LIN {X 0,Y 474.637,Z 525.358,A -85,B 0,C 180,E1 -7446.642,E2 -7446.642} C_VEL
LIN {X 0,Y 474.66,Z 525.36,A -85,B 0,C 180,E1 -7450.09,E2 -7450.09} C_VEL
LIN {X 0,Y 474.663,Z 525.362,A -85,B 0,C 180,E1 -7451.685,E2 -7451.685} C_VEL
LIN {X 0,Y 474.409,Z 525.922,A -85,B 0,C 180,E1 -7452.155,E2 -7452.155} C_VEL
LIN {X 0,Y 473.767,Z 527.315,A -85,B 0,C 180,E1 -7452.599,E2 -7452.599} C_VEL
LIN {X 0,Y 471.839,Z 531.346,A -85,B 0,C 180,E1 -7453.425,E2 -7453.425} C_VEL
LIN {X 0,Y 469.145,Z 537.57,A -85,B 0,C 180,E1 -7454.637,E2 -7454.637} C_VEL
LIN {X 0,Y 468.823,Z 539.587,A -85,B 0,C 180,E1 -7455.057,E2 -7455.057} C_VEL
LIN {X 0,Y 468.432,Z 549.198,A -85,B 0,C 180,E1 -7457.076,E2 -7457.076} C_VEL
LIN {X 0,Y 471.299,Z 564.47,A -85,B 0,C 180,E1 -7457.416,E2 -7457.416} C_VEL
LIN {X 0,Y 470.623,Z 655.993,A -85,B 0,C 180,E1 -7458.833,E2 -7458.833} C_VEL
LIN {X 0,Y 470.332,Z 669.115,A -85,B 0,C 180,E1 -7459.208,E2 -7459.208} C_VEL
LIN {X 0,Y 469.953,Z 682.277,A -85,B 0,C 180,E1 -7459.771,E2 -7459.771} C_VEL
LIN {X 0,Y 469.539,Z 693.349,A -85,B 0,C 180,E1 -7460.415,E2 -7460.415} C_VEL
LIN {X 0,Y 469.046,Z 704.84,A -85,B 0,C 180,E1 -7461.274,E2 -7461.274} C_VEL
LIN {X 0,Y 468.398,Z 715.201,A -85,B 0,C 180,E1 -7462.239,E2 -7462.239} C_VEL
LIN {X 0,Y 468.084,Z 724.517,A -85,B 0,C 180,E1 -7463.318,E2 -7463.318} C_VEL
LIN {X 0,Y 467.692,Z 733.507,A -85,B 0,C 180,E1 -7464.611,E2 -7464.611} C_VEL
LIN {X 0,Y 467.321,Z 740.766,A -85,B 0,C 180,E1 -7465.904,E2 -7465.904} C_VEL
LIN {X 0,Y 466.914,Z 747.443,A -85,B 0,C 180,E1 -7467.412,E2 -7467.412} C_VEL
LIN {X 0,Y 466.79,Z 751.849,A -85,B 0,C 180,E1 -7468.706,E2 -7468.706} C_VEL
LIN {X 0,Y 466.624,Z 755.204,A -85,B 0,C 180,E1 -7470,E2 -7470} C_VEL
LIN {X 0,Y 466.635,Z 758.138,A -85,B 0,C 180,E1 -7471.726,E2 -7471.726} C_VEL
LIN {X 0,Y 466.675,Z 759.019,A -85,B 0,C 180,E1 -7472.589,E2 -7472.589} C_VEL
LIN {X 0,Y 466.669,Z 759.482,A -85,B 0,C 180,E1 -7473.453,E2 -7473.453} C_VEL
LIN {X 0,Y 466.645,Z 759.223,A -85,B 0,C 180,E1 -7475.184,E2 -7475.184} C_VEL
LIN {X 0,Y 466.7,Z 758.184,A -85,B 0,C 180,E1 -7476.334,E2 -7476.334} C_VEL
LIN {X 0,Y 466.711,Z 755.837,A -85,B 0,C 180,E1 -7477.789,E2 -7477.789} C_VEL
LIN {X 0,Y 466.772,Z 752.704,A -85,B 0,C 180,E1 -7479.096,E2 -7479.096} C_VEL
LIN {X 0,Y 466.956,Z 748.499,A -85,B 0,C 180,E1 -7480.405,E2 -7480.405} C_VEL
LIN {X 0,Y 467.201,Z 743.197,A -85,B 0,C 180,E1 -7481.695,E2 -7481.695} C_VEL
LIN {X 0,Y 467.458,Z 736.313,A -85,B 0,C 180,E1 -7483.033,E2 -7483.033} C_VEL
LIN {X 0,Y 467.881,Z 727.842,A -85,B 0,C 180,E1 -7484.35,E2 -7484.35} C_VEL
LIN {X 0,Y 468.362,Z 719.087,A -85,B 0,C 180,E1 -7485.447,E2 -7485.447} C_VEL
LIN {X 0,Y 468.849,Z 708.273,A -85,B 0,C 180,E1 -7486.547,E2 -7486.547} C_VEL
LIN {X 0,Y 469.357,Z 697.427,A -85,B 0,C 180,E1 -7487.426,E2 -7487.426} C_VEL
LIN {X 0,Y 469.888,Z 685.205,A -85,B 0,C 180,E1 -7488.193,E2 -7488.193} C_VEL
LIN {X 0,Y 470.308,Z 672.366,A -85,B 0,C 180,E1 -7488.797,E2 -7488.797} C_VEL
LIN {X 0,Y 470.605,Z 659.785,A -85,B 0,C 180,E1 -7489.201,E2 -7489.201} C_VEL
LIN {X 0,Y 470.83,Z 643.66,A -85,B 0,C 180,E1 -7489.498,E2 -7489.498} C_VEL
LIN {X 0,Y 471.293,Z 563.604,A -85,B 0,C 180,E1 -7490.733,E2 -7490.733} C_VEL
LIN {X 0,Y 468.482,Z 549.194,A -85,B 0,C 180,E1 -7491.071,E2 -7491.071} C_VEL
LIN {X 0,Y 469.083,Z 535.764,A -85,B 0,C 180,E1 -7493.945,E2 -7493.945} C_VEL
LIN {X 0,Y 468.346,Z 529.947,A -85,B 0,C 180,E1 -7495.265,E2 -7495.265} C_VEL
LIN {X 0,Y 467.654,Z 526.235,A -85,B 0,C 180,E1 -7496.136,E2 -7496.136} C_VEL
LIN {X 0,Y 467.571,Z 526.242,A -85,B 0,C 180,E1 -7499.332,E2 -7499.332} C_VEL
LIN {X 0,Y 467.582,Z 526.244,A -85,B 0,C 180,E1 -7502.678,E2 -7502.678} C_VEL
LIN {X 0,Y 467.561,Z 526.241,A -85,B 0,C 180,E1 -7505.739,E2 -7505.739} C_VEL
LIN {X 0,Y 467.614,Z 526.237,A -85,B 0,C 180,E1 -7509.14,E2 -7509.14} C_VEL
LIN {X 0,Y 467.617,Z 526.239,A -85,B 0,C 180,E1 -7512.57,E2 -7512.57} C_VEL
LIN {X 0,Y 467.563,Z 526.241,A -85,B 0,C 180,E1 -7516.176,E2 -7516.176} C_VEL
LIN {X 0,Y 467.578,Z 526.237,A -85,B 0,C 180,E1 -7518.722,E2 -7518.722} C_VEL
LIN {X 0,Y 467.562,Z 526.24,A -85,B 0,C 180,E1 -7521.955,E2 -7521.955} C_VEL
LIN {X 0,Y 467.563,Z 526.24,A -85,B 0,C 180,E1 -7525.167,E2 -7525.167} C_VEL
LIN {X 0,Y 467.579,Z 526.24,A -85,B 0,C 180,E1 -7528.259,E2 -7528.259} C_VEL
LIN {X 0,Y 467.576,Z 526.239,A -85,B 0,C 180,E1 -7531.25,E2 -7531.25} C_VEL
LIN {X 0,Y 467.604,Z 526.233,A -85,B 0,C 180,E1 -7534.159,E2 -7534.159} C_VEL
LIN {X 0,Y 467.569,Z 526.238,A -85,B 0,C 180,E1 -7536.995,E2 -7536.995} C_VEL
LIN {X 0,Y 467.616,Z 526.233,A -85,B 0,C 180,E1 -7539.777,E2 -7539.777} C_VEL
LIN {X 0,Y 467.601,Z 526.237,A -85,B 0,C 180,E1 -7542.506,E2 -7542.506} C_VEL
LIN {X 0,Y 467.597,Z 526.236,A -85,B 0,C 180,E1 -7545.196,E2 -7545.196} C_VEL
LIN {X 0,Y 467.647,Z 526.225,A -85,B 0,C 180,E1 -7547.854,E2 -7547.854} C_VEL
LIN {X 0,Y 467.673,Z 526.224,A -85,B 0,C 180,E1 -7551.357,E2 -7551.357} C_VEL
LIN {X 0,Y 467.738,Z 526.217,A -85,B 0,C 180,E1 -7553.962,E2 -7553.962} C_VEL
LIN {X 0,Y 467.851,Z 526.199,A -85,B 0,C 180,E1 -7557.417,E2 -7557.417} C_VEL
LIN {X 0,Y 467.873,Z 526.201,A -85,B 0,C 180,E1 -7560,E2 -7560} C_VEL
LIN {X 0,Y 467.851,Z 526.206,A -85,B 0,C 180,E1 -7562.583,E2 -7562.583} C_VEL
LIN {X 0,Y 467.734,Z 526.219,A -85,B 0,C 180,E1 -7566.037,E2 -7566.037} C_VEL
LIN {X 0,Y 467.673,Z 526.228,A -85,B 0,C 180,E1 -7568.643,E2 -7568.643} C_VEL
LIN {X 0,Y 467.647,Z 526.231,A -85,B 0,C 180,E1 -7572.146,E2 -7572.146} C_VEL
LIN {X 0,Y 467.63,Z 526.231,A -85,B 0,C 180,E1 -7575.695,E2 -7575.695} C_VEL
LIN {X 0,Y 467.609,Z 526.238,A -85,B 0,C 180,E1 -7578.765,E2 -7578.765} C_VEL
LIN {X 0,Y 467.572,Z 526.238,A -85,B 0,C 180,E1 -7581.269,E2 -7581.269} C_VEL
LIN {X 0,Y 467.564,Z 526.238,A -85,B 0,C 180,E1 -7583.944,E2 -7583.944} C_VEL
LIN {X 0,Y 467.62,Z 526.234,A -85,B 0,C 180,E1 -7586.8,E2 -7586.8} C_VEL
LIN {X 0,Y 467.58,Z 526.237,A -85,B 0,C 180,E1 -7589.736,E2 -7589.736} C_VEL
LIN {X 0,Y 467.577,Z 526.243,A -85,B 0,C 180,E1 -7592.759,E2 -7592.759} C_VEL
LIN {X 0,Y 467.55,Z 526.242,A -85,B 0,C 180,E1 -7595.89,E2 -7595.89} C_VEL
LIN {X 0,Y 467.609,Z 526.235,A -85,B 0,C 180,E1 -7599.142,E2 -7599.142} C_VEL
LIN {X 0,Y 467.581,Z 526.245,A -85,B 0,C 180,E1 -7602.568,E2 -7602.568} C_VEL
LIN {X 0,Y 467.566,Z 526.242,A -85,B 0,C 180,E1 -7605.054,E2 -7605.054} C_VEL
LIN {X 0,Y 467.585,Z 526.238,A -85,B 0,C 180,E1 -7607.441,E2 -7607.441} C_VEL
LIN {X 0,Y 467.58,Z 526.242,A -85,B 0,C 180,E1 -7610.856,E2 -7610.856} C_VEL
LIN {X 0,Y 467.558,Z 526.245,A -85,B 0,C 180,E1 -7614.261,E2 -7614.261} C_VEL
LIN {X 0,Y 467.581,Z 526.239,A -85,B 0,C 180,E1 -7617.321,E2 -7617.321} C_VEL
LIN {X 0,Y 467.57,Z 526.245,A -85,B 0,C 180,E1 -7620.668,E2 -7620.668} C_VEL
LIN {X 0,Y 467.617,Z 526.239,A -85,B 0,C 180,E1 -7623.2,E2 -7623.2} C_VEL
LIN {X 0,Y 467.646,Z 526.388,A -85,B 0,C 180,E1 -7624.163,E2 -7624.163} C_VEL
LIN {X 0,Y 469.844,Z 537.694,A -85,B 0,C 180,E1 -7626.414,E2 -7626.414} C_VEL
LIN {X 0,Y 469.725,Z 543.974,A -85,B 0,C 180,E1 -7627.572,E2 -7627.572} C_VEL
LIN {X 0,Y 468.986,Z 560.3,A -85,B 0,C 180,E1 -7630.524,E2 -7630.524} C_VEL
LIN {X 0,Y 468.438,Z 574.152,A -85,B 0,C 180,E1 -7632.964,E2 -7632.964} C_VEL
LIN {X 0,Y 471.329,Z 593.265,A -85,B 0,C 180,E1 -7633.375,E2 -7633.375} C_VEL
LIN {X 0,Y 470.645,Z 682.622,A -85,B 0,C 180,E1 -7634.769,E2 -7634.769} C_VEL
LIN {X 0,Y 470.151,Z 696.457,A -85,B 0,C 180,E1 -7635.168,E2 -7635.168} C_VEL
LIN {X 0,Y 469.77,Z 708.857,A -85,B 0,C 180,E1 -7635.709,E2 -7635.709} C_VEL
LIN {X 0,Y 469.258,Z 720.253,A -85,B 0,C 180,E1 -7636.379,E2 -7636.379} C_VEL
LIN {X 0,Y 468.795,Z 730.946,A -85,B 0,C 180,E1 -7637.178,E2 -7637.178} C_VEL
LIN {X 0,Y 468.296,Z 741.911,A -85,B 0,C 180,E1 -7638.201,E2 -7638.201} C_VEL
LIN {X 0,Y 467.82,Z 750.431,A -85,B 0,C 180,E1 -7639.177,E2 -7639.177} C_VEL
LIN {X 0,Y 467.477,Z 758.299,A -85,B 0,C 180,E1 -7640.263,E2 -7640.263} C_VEL
LIN {X 0,Y 467.13,Z 765.987,A -85,B 0,C 180,E1 -7641.565,E2 -7641.565} C_VEL
LIN {X 0,Y 466.859,Z 773.081,A -85,B 0,C 180,E1 -7643.083,E2 -7643.083} C_VEL
LIN {X 0,Y 466.783,Z 777.804,A -85,B 0,C 180,E1 -7644.384,E2 -7644.384} C_VEL
LIN {X 0,Y 466.652,Z 781.411,A -85,B 0,C 180,E1 -7645.682,E2 -7645.682} C_VEL
LIN {X 0,Y 466.691,Z 783.275,A -85,B 0,C 180,E1 -7646.547,E2 -7646.547} C_VEL
LIN {X 0,Y 466.662,Z 784.672,A -85,B 0,C 180,E1 -7647.411,E2 -7647.411} C_VEL
LIN {X 0,Y 466.618,Z 786.278,A -85,B 0,C 180,E1 -7649.137,E2 -7649.137} C_VEL
LIN {X 0,Y 466.598,Z 786.495,A -85,B 0,C 180,E1 -7650,E2 -7650} C_VEL
LIN {X 0,Y 466.618,Z 786.28,A -85,B 0,C 180,E1 -7650.863,E2 -7650.863} C_VEL
LIN {X 0,Y 466.662,Z 784.68,A -85,B 0,C 180,E1 -7652.589,E2 -7652.589} C_VEL
LIN {X 0,Y 466.691,Z 783.285,A -85,B 0,C 180,E1 -7653.453,E2 -7653.453} C_VEL
LIN {X 0,Y 466.695,Z 780.348,A -85,B 0,C 180,E1 -7654.751,E2 -7654.751} C_VEL
LIN {X 0,Y 466.781,Z 776.373,A -85,B 0,C 180,E1 -7656.05,E2 -7656.05} C_VEL
LIN {X 0,Y 466.979,Z 770.257,A -85,B 0,C 180,E1 -7657.567,E2 -7657.567} C_VEL
LIN {X 0,Y 467.241,Z 763.572,A -85,B 0,C 180,E1 -7658.869,E2 -7658.869} C_VEL
LIN {X 0,Y 467.593,Z 755.275,A -85,B 0,C 180,E1 -7660.172,E2 -7660.172} C_VEL
LIN {X 0,Y 468.036,Z 746.766,A -85,B 0,C 180,E1 -7661.257,E2 -7661.257} C_VEL
LIN {X 0,Y 468.567,Z 736.518,A -85,B 0,C 180,E1 -7662.316,E2 -7662.316} C_VEL
LIN {X 0,Y 469.014,Z 726.124,A -85,B 0,C 180,E1 -7663.187,E2 -7663.187} C_VEL
LIN {X 0,Y 469.5,Z 714.408,A -85,B 0,C 180,E1 -7663.967,E2 -7663.967} C_VEL
LIN {X 0,Y 469.956,Z 702.633,A -85,B 0,C 180,E1 -7664.561,E2 -7664.561} C_VEL
LIN {X 0,Y 470.343,Z 689.041,A -85,B 0,C 180,E1 -7665.047,E2 -7665.047} C_VEL
LIN {X 0,Y 470.62,Z 676.972,A -85,B 0,C 180,E1 -7665.315,E2 -7665.315} C_VEL
LIN {X 0,Y 471.208,Z 591.98,A -85,B 0,C 180,E1 -7666.614,E2 -7666.614} C_VEL
LIN {X 0,Y 468.379,Z 573.863,A -85,B 0,C 180,E1 -7667.013,E2 -7667.013} C_VEL
LIN {X 0,Y 468.989,Z 557.402,A -85,B 0,C 180,E1 -7669.932,E2 -7669.932} C_VEL
LIN {X 0,Y 469.871,Z 539.602,A -85,B 0,C 180,E1 -7673.118,E2 -7673.118} C_VEL
LIN {X 0,Y 469.298,Z 534.905,A -85,B 0,C 180,E1 -7674.005,E2 -7674.005} C_VEL
LIN {X 0,Y 467.66,Z 526.234,A -85,B 0,C 180,E1 -7675.717,E2 -7675.717} C_VEL
LIN {X 0,Y 467.576,Z 526.241,A -85,B 0,C 180,E1 -7678.749,E2 -7678.749} C_VEL
LIN {X 0,Y 467.583,Z 526.241,A -85,B 0,C 180,E1 -7681.739,E2 -7681.739} C_VEL
LIN {X 0,Y 467.563,Z 526.24,A -85,B 0,C 180,E1 -7684.832,E2 -7684.832} C_VEL
LIN {X 0,Y 467.563,Z 526.24,A -85,B 0,C 180,E1 -7688.044,E2 -7688.044} C_VEL
LIN {X 0,Y 467.578,Z 526.242,A -85,B 0,C 180,E1 -7691.277,E2 -7691.277} C_VEL
LIN {X 0,Y 467.562,Z 526.242,A -85,B 0,C 180,E1 -7693.822,E2 -7693.822} C_VEL
LIN {X 0,Y 467.551,Z 526.24,A -85,B 0,C 180,E1 -7696.255,E2 -7696.255} C_VEL
LIN {X 0,Y 467.579,Z 526.237,A -85,B 0,C 180,E1 -7698.722,E2 -7698.722} C_VEL
LIN {X 0,Y 467.569,Z 526.246,A -85,B 0,C 180,E1 -7701.406,E2 -7701.406} C_VEL
LIN {X 0,Y 467.557,Z 526.24,A -85,B 0,C 180,E1 -7704.26,E2 -7704.26} C_VEL
LIN {X 0,Y 467.575,Z 526.243,A -85,B 0,C 180,E1 -7707.32,E2 -7707.32} C_VEL
LIN {X 0,Y 467.571,Z 526.238,A -85,B 0,C 180,E1 -7710.665,E2 -7710.665} C_VEL
LIN {X 0,Y 467.62,Z 526.236,A -85,B 0,C 180,E1 -7713.2,E2 -7713.2} C_VEL
LIN {X 0,Y 467.584,Z 526.236,A -85,B 0,C 180,E1 -7716.468,E2 -7716.468} C_VEL
LIN {X 0,Y 467.615,Z 526.236,A -85,B 0,C 180,E1 -7719.777,E2 -7719.777} C_VEL
LIN {X 0,Y 467.6,Z 526.234,A -85,B 0,C 180,E1 -7722.506,E2 -7722.506} C_VEL
LIN {X 0,Y 467.6,Z 526.239,A -85,B 0,C 180,E1 -7725.196,E2 -7725.196} C_VEL
LIN {X 0,Y 467.647,Z 526.231,A -85,B 0,C 180,E1 -7727.854,E2 -7727.854} C_VEL
LIN {X 0,Y 467.673,Z 526.232,A -85,B 0,C 180,E1 -7731.357,E2 -7731.357} C_VEL
LIN {X 0,Y 467.734,Z 526.219,A -85,B 0,C 180,E1 -7733.963,E2 -7733.963} C_VEL
LIN {X 0,Y 467.851,Z 526.211,A -85,B 0,C 180,E1 -7737.417,E2 -7737.417} C_VEL
LIN {X 0,Y 467.872,Z 526.202,A -85,B 0,C 180,E1 -7740,E2 -7740} C_VEL
LIN {X 0,Y 467.851,Z 526.203,A -85,B 0,C 180,E1 -7742.583,E2 -7742.583} C_VEL
LIN {X 0,Y 467.742,Z 526.217,A -85,B 0,C 180,E1 -7746.038,E2 -7746.038} C_VEL
LIN {X 0,Y 467.673,Z 526.225,A -85,B 0,C 180,E1 -7748.643,E2 -7748.643} C_VEL
LIN {X 0,Y 467.647,Z 526.229,A -85,B 0,C 180,E1 -7752.146,E2 -7752.146} C_VEL
LIN {X 0,Y 467.63,Z 526.235,A -85,B 0,C 180,E1 -7755.695,E2 -7755.695} C_VEL
LIN {X 0,Y 467.609,Z 526.234,A -85,B 0,C 180,E1 -7758.765,E2 -7758.765} C_VEL
LIN {X 0,Y 467.573,Z 526.244,A -85,B 0,C 180,E1 -7761.269,E2 -7761.269} C_VEL
LIN {X 0,Y 467.565,Z 526.24,A -85,B 0,C 180,E1 -7763.944,E2 -7763.944} C_VEL
LIN {X 0,Y 467.62,Z 526.233,A -85,B 0,C 180,E1 -7766.8,E2 -7766.8} C_VEL
LIN {X 0,Y 467.581,Z 526.24,A -85,B 0,C 180,E1 -7769.737,E2 -7769.737} C_VEL
LIN {X 0,Y 467.578,Z 526.238,A -85,B 0,C 180,E1 -7772.759,E2 -7772.759} C_VEL
LIN {X 0,Y 467.551,Z 526.242,A -85,B 0,C 180,E1 -7775.89,E2 -7775.89} C_VEL
LIN {X 0,Y 467.578,Z 526.241,A -85,B 0,C 180,E1 -7779.146,E2 -7779.146} C_VEL
LIN {X 0,Y 467.582,Z 526.236,A -85,B 0,C 180,E1 -7782.568,E2 -7782.568} C_VEL
LIN {X 0,Y 467.567,Z 526.242,A -85,B 0,C 180,E1 -7785.054,E2 -7785.054} C_VEL
LIN {X 0,Y 467.622,Z 526.239,A -85,B 0,C 180,E1 -7787.445,E2 -7787.445} C_VEL
LIN {X 0,Y 467.614,Z 526.234,A -85,B 0,C 180,E1 -7790.86,E2 -7790.86} C_VEL
LIN {X 0,Y 467.561,Z 526.239,A -85,B 0,C 180,E1 -7794.261,E2 -7794.261} C_VEL
LIN {X 0,Y 467.582,Z 526.244,A -85,B 0,C 180,E1 -7797.322,E2 -7797.322} C_VEL
LIN {X 0,Y 467.571,Z 526.238,A -85,B 0,C 180,E1 -7800.668,E2 -7800.668} C_VEL
LIN {X 0,Y 467.618,Z 526.237,A -85,B 0,C 180,E1 -7803.201,E2 -7803.201} C_VEL
LIN {X 0,Y 467.594,Z 526.234,A -85,B 0,C 180,E1 -7806.469,E2 -7806.469} C_VEL
LIN {X 0,Y 467.627,Z 526.239,A -85,B 0,C 180,E1 -7809.778,E2 -7809.778} C_VEL
LIN {X 0,Y 467.65,Z 526.283,A -85,B 0,C 180,E1 -7812.113,E2 -7812.113} C_VEL
LIN {X 0,Y 468.98,Z 534.562,A -85,B 0,C 180,E1 -7813.982,E2 -7813.982} C_VEL
LIN {X 0,Y 468.823,Z 539.587,A -85,B 0,C 180,E1 -7815.057,E2 -7815.057} C_VEL
LIN {X 0,Y 468.19,Z 542.859,A -85,B 0,C 180,E1 -7815.631,E2 -7815.631} C_VEL
LIN {X 0,Y 466.408,Z 548.22,A -85,B 0,C 180,E1 -7816.276,E2 -7816.276} C_VEL
LIN {X 0,Y 464.654,Z 554.481,A -85,B 0,C 180,E1 -7816.775,E2 -7816.775} C_VEL
LIN {X 0,Y 464.025,Z 559.712,A -85,B 0,C 180,E1 -7817.039,E2 -7817.039} C_VEL
LIN {X 0,Y 464.238,Z 563.371,A -85,B 0,C 180,E1 -7817.149,E2 -7817.149} C_VEL
LIN {X 0,Y 464.487,Z 568.128,A -85,B 0,C 180,E1 -7817.233,E2 -7817.233} C_VEL
LIN {X 0,Y 463.775,Z 655.979,A -85,B 0,C 180,E1 -7818.611,E2 -7818.611} C_VEL
LIN {X 0,Y 463.466,Z 669.181,A -85,B 0,C 180,E1 -7818.991,E2 -7818.991} C_VEL
LIN {X 0,Y 463.074,Z 682.388,A -85,B 0,C 180,E1 -7819.562,E2 -7819.562} C_VEL
LIN {X 0,Y 462.6,Z 694.274,A -85,B 0,C 180,E1 -7820.27,E2 -7820.27} C_VEL
LIN {X 0,Y 462.075,Z 705.637,A -85,B 0,C 180,E1 -7821.142,E2 -7821.142} C_VEL
LIN {X 0,Y 461.415,Z 715.898,A -85,B 0,C 180,E1 -7822.121,E2 -7822.121} C_VEL
LIN {X 0,Y 461.074,Z 725.105,A -85,B 0,C 180,E1 -7823.216,E2 -7823.216} C_VEL
LIN {X 0,Y 460.654,Z 734.032,A -85,B 0,C 180,E1 -7824.528,E2 -7824.528} C_VEL
LIN {X 0,Y 460.282,Z 741.236,A -85,B 0,C 180,E1 -7825.841,E2 -7825.841} C_VEL
LIN {X 0,Y 459.846,Z 747.841,A -85,B 0,C 180,E1 -7827.372,E2 -7827.372} C_VEL
LIN {X 0,Y 459.708,Z 752.204,A -85,B 0,C 180,E1 -7828.686,E2 -7828.686} C_VEL
LIN {X 0,Y 459.554,Z 755.517,A -85,B 0,C 180,E1 -7830,E2 -7830} C_VEL
LIN {X 0,Y 459.556,Z 757.162,A -85,B 0,C 180,E1 -7830.876,E2 -7830.876} C_VEL
LIN {X 0,Y 459.595,Z 759.268,A -85,B 0,C 180,E1 -7832.629,E2 -7832.629} C_VEL
LIN {X 0,Y 459.564,Z 759.697,A -85,B 0,C 180,E1 -7833.507,E2 -7833.507} C_VEL
LIN {X 0,Y 459.555,Z 759.398,A -85,B 0,C 180,E1 -7835.265,E2 -7835.265} C_VEL
LIN {X 0,Y 459.594,Z 758.495,A -85,B 0,C 180,E1 -7836.295,E2 -7836.295} C_VEL
LIN {X 0,Y 459.634,Z 755.932,A -85,B 0,C 180,E1 -7837.91,E2 -7837.91} C_VEL
LIN {X 0,Y 459.7,Z 752.758,A -85,B 0,C 180,E1 -7839.237,E2 -7839.237} C_VEL
LIN {X 0,Y 459.894,Z 748.508,A -85,B 0,C 180,E1 -7840.567,E2 -7840.567} C_VEL
LIN {X 0,Y 460.147,Z 743.387,A -85,B 0,C 180,E1 -7841.826,E2 -7841.826} C_VEL
LIN {X 0,Y 460.46,Z 736.224,A -85,B 0,C 180,E1 -7843.235,E2 -7843.235} C_VEL
LIN {X 0,Y 460.841,Z 729.229,A -85,B 0,C 180,E1 -7844.348,E2 -7844.348} C_VEL
LIN {X 0,Y 461.324,Z 720.78,A -85,B 0,C 180,E1 -7845.462,E2 -7845.462} C_VEL
LIN {X 0,Y 461.792,Z 711.089,A -85,B 0,C 180,E1 -7846.504,E2 -7846.504} C_VEL
LIN {X 0,Y 462.342,Z 699.888,A -85,B 0,C 180,E1 -7847.47,E2 -7847.47} C_VEL
LIN {X 0,Y 462.911,Z 688.453,A -85,B 0,C 180,E1 -7848.248,E2 -7848.248} C_VEL
LIN {X 0,Y 463.372,Z 676.645,A -85,B 0,C 180,E1 -7848.859,E2 -7848.859} C_VEL
LIN {X 0,Y 463.691,Z 664.781,A -85,B 0,C 180,E1 -7849.305,E2 -7849.305} C_VEL
LIN {X 0,Y 463.928,Z 650.899,A -85,B 0,C 180,E1 -7849.635,E2 -7849.635} C_VEL
LIN {X 0,Y 464.54,Z 564.559,A -85,B 0,C 180,E1 -7850.985,E2 -7850.985} C_VEL
LIN {X 0,Y 461.587,Z 549.362,A -85,B 0,C 180,E1 -7851.357,E2 -7851.357} C_VEL
LIN {X 0,Y 462.081,Z 536.091,A -85,B 0,C 180,E1 -7854.245,E2 -7854.245} C_VEL
LIN {X 0,Y 460.991,Z 528.936,A -85,B 0,C 180,E1 -7855.909,E2 -7855.909} C_VEL
LIN {X 0,Y 460.599,Z 527.115,A -85,B 0,C 180,E1 -7856.384,E2 -7856.384} C_VEL
LIN {X 0,Y 460.532,Z 527.118,A -85,B 0,C 180,E1 -7859.558,E2 -7859.558} C_VEL
LIN {X 0,Y 460.531,Z 527.12,A -85,B 0,C 180,E1 -7862.283,E2 -7862.283} C_VEL
LIN {X 0,Y 460.512,Z 527.119,A -85,B 0,C 180,E1 -7865.444,E2 -7865.444} C_VEL
LIN {X 0,Y 460.565,Z 527.118,A -85,B 0,C 180,E1 -7868.9,E2 -7868.9} C_VEL
LIN {X 0,Y 460.546,Z 527.115,A -85,B 0,C 180,E1 -7872.178,E2 -7872.178} C_VEL
LIN {X 0,Y 460.517,Z 527.117,A -85,B 0,C 180,E1 -7875.411,E2 -7875.411} C_VEL
LIN {X 0,Y 460.531,Z 527.117,A -85,B 0,C 180,E1 -7878.396,E2 -7878.396} C_VEL
LIN {X 0,Y 460.526,Z 527.118,A -85,B 0,C 180,E1 -7881.267,E2 -7881.267} C_VEL
LIN {X 0,Y 460.508,Z 527.124,A -85,B 0,C 180,E1 -7884.554,E2 -7884.554} C_VEL
LIN {X 0,Y 460.526,Z 527.116,A -85,B 0,C 180,E1 -7887.715,E2 -7887.715} C_VEL
LIN {X 0,Y 460.541,Z 527.121,A -85,B 0,C 180,E1 -7890.769,E2 -7890.769} C_VEL
LIN {X 0,Y 460.561,Z 527.108,A -85,B 0,C 180,E1 -7893.734,E2 -7893.734} C_VEL
LIN {X 0,Y 460.538,Z 527.119,A -85,B 0,C 180,E1 -7896.623,E2 -7896.623} C_VEL
LIN {X 0,Y 460.544,Z 527.114,A -85,B 0,C 180,E1 -7899.452,E2 -7899.452} C_VEL
LIN {X 0,Y 460.551,Z 527.113,A -85,B 0,C 180,E1 -7902.23,E2 -7902.23} C_VEL
LIN {X 0,Y 460.556,Z 527.115,A -85,B 0,C 180,E1 -7904.964,E2 -7904.964} C_VEL
LIN {X 0,Y 460.604,Z 527.11,A -85,B 0,C 180,E1 -7908.559,E2 -7908.559} C_VEL
LIN {X 0,Y 460.686,Z 527.095,A -85,B 0,C 180,E1 -7912.108,E2 -7912.108} C_VEL
LIN {X 0,Y 460.692,Z 527.102,A -85,B 0,C 180,E1 -7914.748,E2 -7914.748} C_VEL
LIN {X 0,Y 460.817,Z 527.075,A -85,B 0,C 180,E1 -7917.377,E2 -7917.377} C_VEL
LIN {X 0,Y 460.844,Z 527.077,A -85,B 0,C 180,E1 -7920,E2 -7920} C_VEL
LIN {X 0,Y 460.816,Z 527.082,A -85,B 0,C 180,E1 -7922.622,E2 -7922.622} C_VEL
LIN {X 0,Y 460.701,Z 527.096,A -85,B 0,C 180,E1 -7926.13,E2 -7926.13} C_VEL
LIN {X 0,Y 460.62,Z 527.107,A -85,B 0,C 180,E1 -7928.776,E2 -7928.776} C_VEL
LIN {X 0,Y 460.604,Z 527.112,A -85,B 0,C 180,E1 -7932.445,E2 -7932.445} C_VEL
LIN {X 0,Y 460.591,Z 527.109,A -85,B 0,C 180,E1 -7935.998,E2 -7935.998} C_VEL
LIN {X 0,Y 460.562,Z 527.114,A -85,B 0,C 180,E1 -7938.902,E2 -7938.902} C_VEL
LIN {X 0,Y 460.507,Z 527.118,A -85,B 0,C 180,E1 -7941.486,E2 -7941.486} C_VEL
LIN {X 0,Y 460.534,Z 527.117,A -85,B 0,C 180,E1 -7944.333,E2 -7944.333} C_VEL
LIN {X 0,Y 460.576,Z 527.107,A -85,B 0,C 180,E1 -7947.244,E2 -7947.244} C_VEL
LIN {X 0,Y 460.52,Z 527.12,A -85,B 0,C 180,E1 -7950.239,E2 -7950.239} C_VEL
LIN {X 0,Y 460.523,Z 527.117,A -85,B 0,C 180,E1 -7953.325,E2 -7953.325} C_VEL
LIN {X 0,Y 460.473,Z 527.129,A -85,B 0,C 180,E1 -7956.53,E2 -7956.53} C_VEL
LIN {X 0,Y 460.57,Z 527.111,A -85,B 0,C 180,E1 -7959.859,E2 -7959.859} C_VEL
LIN {X 0,Y 460.508,Z 527.123,A -85,B 0,C 180,E1 -7962.901,E2 -7962.901} C_VEL
LIN {X 0,Y 460.515,Z 527.119,A -85,B 0,C 180,E1 -7965.83,E2 -7965.83} C_VEL
LIN {X 0,Y 460.53,Z 527.118,A -85,B 0,C 180,E1 -7968.99,E2 -7968.99} C_VEL
LIN {X 0,Y 460.524,Z 527.118,A -85,B 0,C 180,E1 -7971.268,E2 -7971.268} C_VEL
LIN {X 0,Y 460.509,Z 527.123,A -85,B 0,C 180,E1 -7974.555,E2 -7974.555} C_VEL
LIN {X 0,Y 460.531,Z 527.118,A -85,B 0,C 180,E1 -7977.716,E2 -7977.716} C_VEL
LIN {X 0,Y 460.54,Z 527.12,A -85,B 0,C 180,E1 -7980.77,E2 -7980.77} C_VEL
LIN {X 0,Y 460.579,Z 527.115,A -85,B 0,C 180,E1 -7983.736,E2 -7983.736} C_VEL
LIN {X 0,Y 460.601,Z 527.356,A -85,B 0,C 180,E1 -7983.937,E2 -7983.937} C_VEL
LIN {X 0,Y 462.891,Z 538.877,A -85,B 0,C 180,E1 -7986.276,E2 -7986.276} C_VEL
LIN {X 0,Y 462.91,Z 543.898,A -85,B 0,C 180,E1 -7987.224,E2 -7987.224} C_VEL
LIN {X 0,Y 462.008,Z 561.451,A -85,B 0,C 180,E1 -7990.449,E2 -7990.449} C_VEL
LIN {X 0,Y 461.469,Z 573.846,A -85,B 0,C 180,E1 -7992.682,E2 -7992.682} C_VEL
LIN {X 0,Y 464.568,Z 593.927,A -85,B 0,C 180,E1 -7993.126,E2 -7993.126} C_VEL
LIN {X 0,Y 463.845,Z 681.794,A -85,B 0,C 180,E1 -7994.512,E2 -7994.512} C_VEL
LIN {X 0,Y 463.38,Z 695.068,A -85,B 0,C 180,E1 -7994.89,E2 -7994.89} C_VEL
LIN {X 0,Y 462.939,Z 707.788,A -85,B 0,C 180,E1 -7995.438,E2 -7995.438} C_VEL
LIN {X 0,Y 462.36,Z 719.897,A -85,B 0,C 180,E1 -7996.149,E2 -7996.149} C_VEL
LIN {X 0,Y 461.804,Z 731.807,A -85,B 0,C 180,E1 -7997.062,E2 -7997.062} C_VEL
LIN {X 0,Y 461.265,Z 742.836,A -85,B 0,C 180,E1 -7998.13,E2 -7998.13} C_VEL
LIN {X 0,Y 460.749,Z 751.971,A -85,B 0,C 180,E1 -7999.231,E2 -7999.231} C_VEL
LIN {X 0,Y 460.324,Z 760.884,A -85,B 0,C 180,E1 -8000.554,E2 -8000.554} C_VEL
LIN {X 0,Y 460.007,Z 768.06,A -85,B 0,C 180,E1 -8001.876,E2 -8001.876} C_VEL
LIN {X 0,Y 459.746,Z 774.068,A -85,B 0,C 180,E1 -8003.273,E2 -8003.273} C_VEL
LIN {X 0,Y 459.661,Z 778.929,A -85,B 0,C 180,E1 -8004.737,E2 -8004.737} C_VEL
LIN {X 0,Y 459.57,Z 781.221,A -85,B 0,C 180,E1 -8005.615,E2 -8005.615} C_VEL
LIN {X 0,Y 459.586,Z 783.081,A -85,B 0,C 180,E1 -8006.493,E2 -8006.493} C_VEL
LIN {X 0,Y 459.584,Z 784.475,A -85,B 0,C 180,E1 -8007.371,E2 -8007.371} C_VEL
LIN {X 0,Y 459.521,Z 786.076,A -85,B 0,C 180,E1 -8009.124,E2 -8009.124} C_VEL
LIN {X 0,Y 459.53,Z 786.291,A -85,B 0,C 180,E1 -8010,E2 -8010} C_VEL
LIN {X 0,Y 459.521,Z 786.073,A -85,B 0,C 180,E1 -8010.876,E2 -8010.876} C_VEL
LIN {X 0,Y 459.584,Z 784.469,A -85,B 0,C 180,E1 -8012.629,E2 -8012.629} C_VEL
LIN {X 0,Y 459.586,Z 783.07,A -85,B 0,C 180,E1 -8013.507,E2 -8013.507} C_VEL
LIN {X 0,Y 459.623,Z 780.128,A -85,B 0,C 180,E1 -8014.824,E2 -8014.824} C_VEL
LIN {X 0,Y 459.714,Z 775.111,A -85,B 0,C 180,E1 -8016.43,E2 -8016.43} C_VEL
LIN {X 0,Y 459.951,Z 769.004,A -85,B 0,C 180,E1 -8017.904,E2 -8017.904} C_VEL
LIN {X 0,Y 460.241,Z 762.08,A -85,B 0,C 180,E1 -8019.226,E2 -8019.226} C_VEL
LIN {X 0,Y 460.546,Z 755.007,A -85,B 0,C 180,E1 -8020.329,E2 -8020.329} C_VEL
LIN {X 0,Y 461.048,Z 746.478,A -85,B 0,C 180,E1 -8021.429,E2 -8021.429} C_VEL
LIN {X 0,Y 461.581,Z 736.397,A -85,B 0,C 180,E1 -8022.487,E2 -8022.487} C_VEL
LIN {X 0,Y 462.074,Z 725.487,A -85,B 0,C 180,E1 -8023.411,E2 -8023.411} C_VEL
LIN {X 0,Y 462.592,Z 714.015,A -85,B 0,C 180,E1 -8024.18,E2 -8024.18} C_VEL
LIN {X 0,Y 463.076,Z 702.153,A -85,B 0,C 180,E1 -8024.783,E2 -8024.783} C_VEL
LIN {X 0,Y 463.479,Z 688.443,A -85,B 0,C 180,E1 -8025.276,E2 -8025.276} C_VEL
LIN {X 0,Y 463.772,Z 676.111,A -85,B 0,C 180,E1 -8025.547,E2 -8025.547} C_VEL
LIN {X 0,Y 464.262,Z 591.961,A -85,B 0,C 180,E1 -8026.853,E2 -8026.853} C_VEL
LIN {X 0,Y 461.374,Z 573.641,A -85,B 0,C 180,E1 -8027.269,E2 -8027.269} C_VEL
LIN {X 0,Y 462.079,Z 557.124,A -85,B 0,C 180,E1 -8030.243,E2 -8030.243} C_VEL
LIN {X 0,Y 462.922,Z 540.598,A -85,B 0,C 180,E1 -8033.248,E2 -8033.248} C_VEL
LIN {X 0,Y 461.724,Z 532.892,A -85,B 0,C 180,E1 -8034.745,E2 -8034.745} C_VEL
LIN {X 0,Y 460.58,Z 527.115,A -85,B 0,C 180,E1 -8035.925,E2 -8035.925} C_VEL
LIN {X 0,Y 460.555,Z 527.115,A -85,B 0,C 180,E1 -8038.232,E2 -8038.232} C_VEL
LIN {X 0,Y 460.521,Z 527.123,A -85,B 0,C 180,E1 -8041.283,E2 -8041.283} C_VEL
LIN {X 0,Y 460.53,Z 527.115,A -85,B 0,C 180,E1 -8044.505,E2 -8044.505} C_VEL
LIN {X 0,Y 460.525,Z 527.121,A -85,B 0,C 180,E1 -8047.62,E2 -8047.62} C_VEL
LIN {X 0,Y 460.54,Z 527.114,A -85,B 0,C 180,E1 -8050.269,E2 -8050.269} C_VEL
LIN {X 0,Y 460.505,Z 527.125,A -85,B 0,C 180,E1 -8053.373,E2 -8053.373} C_VEL
LIN {X 0,Y 460.495,Z 527.119,A -85,B 0,C 180,E1 -8056.624,E2 -8056.624} C_VEL
LIN {X 0,Y 460.552,Z 527.116,A -85,B 0,C 180,E1 -8059.727,E2 -8059.727} C_VEL
LIN {X 0,Y 460.522,Z 527.116,A -85,B 0,C 180,E1 -8062.518,E2 -8062.518} C_VEL
LIN {X 0,Y 460.542,Z 527.119,A -85,B 0,C 180,E1 -8065.623,E2 -8065.623} C_VEL
LIN {X 0,Y 460.53,Z 527.115,A -85,B 0,C 180,E1 -8068.744,E2 -8068.744} C_VEL
LIN {X 0,Y 460.551,Z 527.116,A -85,B 0,C 180,E1 -8071.767,E2 -8071.767} C_VEL
LIN {X 0,Y 460.551,Z 527.112,A -85,B 0,C 180,E1 -8074.705,E2 -8074.705} C_VEL
LIN {X 0,Y 460.503,Z 527.125,A -85,B 0,C 180,E1 -8077.571,E2 -8077.571} C_VEL
LIN {X 0,Y 460.561,Z 527.111,A -85,B 0,C 180,E1 -8080.384,E2 -8080.384} C_VEL
LIN {X 0,Y 460.556,Z 527.115,A -85,B 0,C 180,E1 -8083.146,E2 -8083.146} C_VEL
LIN {X 0,Y 460.548,Z 527.115,A -85,B 0,C 180,E1 -8085.868,E2 -8085.868} C_VEL
LIN {X 0,Y 460.604,Z 527.105,A -85,B 0,C 180,E1 -8088.559,E2 -8088.559} C_VEL
LIN {X 0,Y 460.685,Z 527.096,A -85,B 0,C 180,E1 -8092.108,E2 -8092.108} C_VEL
LIN {X 0,Y 460.689,Z 527.096,A -85,B 0,C 180,E1 -8094.748,E2 -8094.748} C_VEL
LIN {X 0,Y 460.816,Z 527.087,A -85,B 0,C 180,E1 -8097.378,E2 -8097.378} C_VEL
LIN {X 0,Y 460.843,Z 527.077,A -85,B 0,C 180,E1 -8100,E2 -8100} C_VEL
LIN {X 0,Y 460.817,Z 527.079,A -85,B 0,C 180,E1 -8102.623,E2 -8102.623} C_VEL
LIN {X 0,Y 460.707,Z 527.093,A -85,B 0,C 180,E1 -8106.13,E2 -8106.13} C_VEL
LIN {X 0,Y 460.62,Z 527.104,A -85,B 0,C 180,E1 -8108.776,E2 -8108.776} C_VEL
LIN {X 0,Y 460.604,Z 527.105,A -85,B 0,C 180,E1 -8112.445,E2 -8112.445} C_VEL
LIN {X 0,Y 460.591,Z 527.108,A -85,B 0,C 180,E1 -8115.998,E2 -8115.998} C_VEL
LIN {X 0,Y 460.563,Z 527.112,A -85,B 0,C 180,E1 -8118.902,E2 -8118.902} C_VEL
LIN {X 0,Y 460.508,Z 527.125,A -85,B 0,C 180,E1 -8121.486,E2 -8121.486} C_VEL
LIN {X 0,Y 460.535,Z 527.114,A -85,B 0,C 180,E1 -8124.333,E2 -8124.333} C_VEL
LIN {X 0,Y 460.577,Z 527.115,A -85,B 0,C 180,E1 -8127.244,E2 -8127.244} C_VEL
LIN {X 0,Y 460.521,Z 527.116,A -85,B 0,C 180,E1 -8130.24,E2 -8130.24} C_VEL
LIN {X 0,Y 460.524,Z 527.123,A -85,B 0,C 180,E1 -8133.326,E2 -8133.326} C_VEL
LIN {X 0,Y 460.474,Z 527.122,A -85,B 0,C 180,E1 -8136.53,E2 -8136.53} C_VEL
LIN {X 0,Y 460.554,Z 527.114,A -85,B 0,C 180,E1 -8139.86,E2 -8139.86} C_VEL
LIN {X 0,Y 460.513,Z 527.119,A -85,B 0,C 180,E1 -8142.902,E2 -8142.902} C_VEL
LIN {X 0,Y 460.521,Z 527.118,A -85,B 0,C 180,E1 -8145.83,E2 -8145.83} C_VEL
LIN {X 0,Y 460.541,Z 527.116,A -85,B 0,C 180,E1 -8148.991,E2 -8148.991} C_VEL
LIN {X 0,Y 460.543,Z 527.12,A -85,B 0,C 180,E1 -8151.27,E2 -8151.27} C_VEL
LIN {X 0,Y 460.512,Z 527.117,A -85,B 0,C 180,E1 -8154.555,E2 -8154.555} C_VEL
LIN {X 0,Y 460.531,Z 527.118,A -85,B 0,C 180,E1 -8157.717,E2 -8157.717} C_VEL
LIN {X 0,Y 460.541,Z 527.114,A -85,B 0,C 180,E1 -8160.77,E2 -8160.77} C_VEL
LIN {X 0,Y 460.565,Z 527.114,A -85,B 0,C 180,E1 -8163.736,E2 -8163.736} C_VEL
LIN {X 0,Y 460.548,Z 527.113,A -85,B 0,C 180,E1 -8166.625,E2 -8166.625} C_VEL
LIN {X 0,Y 460.555,Z 527.122,A -85,B 0,C 180,E1 -8169.453,E2 -8169.453} C_VEL
LIN {X 0,Y 460.608,Z 527.19,A -85,B 0,C 180,E1 -8171.945,E2 -8171.945} C_VEL
LIN {X 0,Y 461.971,Z 535.239,A -85,B 0,C 180,E1 -8173.793,E2 -8173.793} C_VEL
LIN {X 0,Y 461.579,Z 547.094,A -85,B 0,C 180,E1 -8176.35,E2 -8176.35} C_VEL
LIN {X 0,Y 461.474,Z 549.302,A -85,B 0,C 180,E1 -8176.819,E2 -8176.819} C_VEL
LIN {X 0,Y 464.238,Z 563.371,A -85,B 0,C 180,E1 -8177.149,E2 -8177.149} C_VEL
LIN {X 0,Y 464.363,Z 567.239,A -85,B 0,C 180,E1 -8177.215,E2 -8177.215} C_VEL
LIN {X 0,Y 463.785,Z 571.104,A -85,B 0,C 180,E1 -8177.255,E2 -8177.255} C_VEL
LIN {X 0,Y 461.42,Z 578.691,A -85,B 0,C 180,E1 -8177.291,E2 -8177.291} C_VEL
LIN {X 0,Y 458.253,Z 588.238,A -85,B 0,C 180,E1 -8177.33,E2 -8177.33} C_VEL
LIN {X 0,Y 457.512,Z 594.139,A -85,B 0,C 180,E1 -8177.398,E2 -8177.398} C_VEL
LIN {X 0,Y 456.904,Z 657.02,A -85,B 0,C 180,E1 -8178.409,E2 -8178.409} C_VEL
LIN {X 0,Y 456.564,Z 670.7,A -85,B 0,C 180,E1 -8178.822,E2 -8178.822} C_VEL
LIN {X 0,Y 456.15,Z 683.496,A -85,B 0,C 180,E1 -8179.402,E2 -8179.402} C_VEL
LIN {X 0,Y 455.655,Z 695.167,A -85,B 0,C 180,E1 -8180.12,E2 -8180.12} C_VEL
LIN {X 0,Y 455.108,Z 706.408,A -85,B 0,C 180,E1 -8181.005,E2 -8181.005} C_VEL
LIN {X 0,Y 454.416,Z 716.565,A -85,B 0,C 180,E1 -8181.999,E2 -8181.999} C_VEL
LIN {X 0,Y 454.065,Z 725.67,A -85,B 0,C 180,E1 -8183.111,E2 -8183.111} C_VEL
LIN {X 0,Y 453.607,Z 734.54,A -85,B 0,C 180,E1 -8184.443,E2 -8184.443} C_VEL
LIN {X 0,Y 453.241,Z 741.691,A -85,B 0,C 180,E1 -8185.776,E2 -8185.776} C_VEL
LIN {X 0,Y 452.949,Z 746.528,A -85,B 0,C 180,E1 -8186.887,E2 -8186.887} C_VEL
LIN {X 0,Y 452.63,Z 751.236,A -85,B 0,C 180,E1 -8188.22,E2 -8188.22} C_VEL
LIN {X 0,Y 452.551,Z 754.841,A -85,B 0,C 180,E1 -8189.555,E2 -8189.555} C_VEL
LIN {X 0,Y 452.461,Z 757.45,A -85,B 0,C 180,E1 -8190.89,E2 -8190.89} C_VEL
LIN {X 0,Y 452.461,Z 758.681,A -85,B 0,C 180,E1 -8191.78,E2 -8191.78} C_VEL
LIN {X 0,Y 452.517,Z 759.507,A -85,B 0,C 180,E1 -8192.67,E2 -8192.67} C_VEL
LIN {X 0,Y 452.432,Z 759.934,A -85,B 0,C 180,E1 -8194.454,E2 -8194.454} C_VEL
LIN {X 0,Y 452.472,Z 759.575,A -85,B 0,C 180,E1 -8195.347,E2 -8195.347} C_VEL
LIN {X 0,Y 452.516,Z 758.768,A -85,B 0,C 180,E1 -8196.286,E2 -8196.286} C_VEL
LIN {X 0,Y 452.551,Z 756.034,A -85,B 0,C 180,E1 -8198.034,E2 -8198.034} C_VEL
LIN {X 0,Y 452.642,Z 752.82,A -85,B 0,C 180,E1 -8199.383,E2 -8199.383} C_VEL
LIN {X 0,Y 452.848,Z 748.529,A -85,B 0,C 180,E1 -8200.733,E2 -8200.733} C_VEL
LIN {X 0,Y 453.134,Z 742.171,A -85,B 0,C 180,E1 -8202.279,E2 -8202.279} C_VEL
LIN {X 0,Y 453.546,Z 734.828,A -85,B 0,C 180,E1 -8203.668,E2 -8203.668} C_VEL
LIN {X 0,Y 454.069,Z 725.868,A -85,B 0,C 180,E1 -8205.025,E2 -8205.025} C_VEL
LIN {X 0,Y 454.652,Z 716.635,A -85,B 0,C 180,E1 -8206.155,E2 -8206.155} C_VEL
LIN {X 0,Y 455.137,Z 706.307,A -85,B 0,C 180,E1 -8207.176,E2 -8207.176} C_VEL
LIN {X 0,Y 455.749,Z 694.82,A -85,B 0,C 180,E1 -8208.079,E2 -8208.079} C_VEL
LIN {X 0,Y 456.33,Z 682.807,A -85,B 0,C 180,E1 -8208.811,E2 -8208.811} C_VEL
LIN {X 0,Y 456.689,Z 670.121,A -85,B 0,C 180,E1 -8209.379,E2 -8209.379} C_VEL
LIN {X 0,Y 457.094,Z 656.316,A -85,B 0,C 180,E1 -8209.787,E2 -8209.787} C_VEL
LIN {X 0,Y 457.91,Z 566.085,A -85,B 0,C 180,E1 -8211.232,E2 -8211.232} C_VEL
LIN {X 0,Y 454.66,Z 549.522,A -85,B 0,C 180,E1 -8211.657,E2 -8211.657} C_VEL
LIN {X 0,Y 455.145,Z 538.835,A -85,B 0,C 180,E1 -8214.009,E2 -8214.009} C_VEL
LIN {X 0,Y 454.683,Z 533.893,A -85,B 0,C 180,E1 -8215.154,E2 -8215.154} C_VEL
LIN {X 0,Y 453.573,Z 527.989,A -85,B 0,C 180,E1 -8216.613,E2 -8216.613} C_VEL
LIN {X 0,Y 453.473,Z 527.998,A -85,B 0,C 180,E1 -8219.784,E2 -8219.784} C_VEL
LIN {X 0,Y 453.49,Z 527.997,A -85,B 0,C 180,E1 -8223.188,E2 -8223.188} C_VEL
LIN {X 0,Y 453.454,Z 528.001,A -85,B 0,C 180,E1 -8226.299,E2 -8226.299} C_VEL
LIN {X 0,Y 453.53,Z 527.989,A -85,B 0,C 180,E1 -8229.444,E2 -8229.444} C_VEL
LIN {X 0,Y 453.49,Z 527.996,A -85,B 0,C 180,E1 -8232.991,E2 -8232.991} C_VEL
LIN {X 0,Y 453.47,Z 527.995,A -85,B 0,C 180,E1 -8235.779,E2 -8235.779} C_VEL
LIN {X 0,Y 453.511,Z 527.986,A -85,B 0,C 180,E1 -8239.405,E2 -8239.405} C_VEL
LIN {X 0,Y 453.469,Z 527.998,A -85,B 0,C 180,E1 -8242.222,E2 -8242.222} C_VEL
LIN {X 0,Y 453.484,Z 527.994,A -85,B 0,C 180,E1 -8245.221,E2 -8245.221} C_VEL
LIN {X 0,Y 453.478,Z 528,A -85,B 0,C 180,E1 -8248.47,E2 -8248.47} C_VEL
LIN {X 0,Y 453.509,Z 527.991,A -85,B 0,C 180,E1 -8251.288,E2 -8251.288} C_VEL
LIN {X 0,Y 453.518,Z 527.989,A -85,B 0,C 180,E1 -8254.284,E2 -8254.284} C_VEL
LIN {X 0,Y 453.471,Z 527.992,A -85,B 0,C 180,E1 -8257.203,E2 -8257.203} C_VEL
LIN {X 0,Y 453.497,Z 527.993,A -85,B 0,C 180,E1 -8260.066,E2 -8260.066} C_VEL
LIN {X 0,Y 453.499,Z 527.995,A -85,B 0,C 180,E1 -8262.875,E2 -8262.875} C_VEL
LIN {X 0,Y 453.504,Z 527.99,A -85,B 0,C 180,E1 -8265.643,E2 -8265.643} C_VEL
LIN {X 0,Y 453.552,Z 527.985,A -85,B 0,C 180,E1 -8268.379,E2 -8268.379} C_VEL
LIN {X 0,Y 453.643,Z 527.972,A -85,B 0,C 180,E1 -8271.985,E2 -8271.985} C_VEL
LIN {X 0,Y 453.666,Z 527.978,A -85,B 0,C 180,E1 -8274.667,E2 -8274.667} C_VEL
LIN {X 0,Y 453.757,Z 527.955,A -85,B 0,C 180,E1 -8277.337,E2 -8277.337} C_VEL
LIN {X 0,Y 453.814,Z 527.952,A -85,B 0,C 180,E1 -8280,E2 -8280} C_VEL
LIN {X 0,Y 453.757,Z 527.96,A -85,B 0,C 180,E1 -8282.663,E2 -8282.663} C_VEL
LIN {X 0,Y 453.668,Z 527.973,A -85,B 0,C 180,E1 -8286.225,E2 -8286.225} C_VEL
LIN {X 0,Y 453.584,Z 527.983,A -85,B 0,C 180,E1 -8288.913,E2 -8288.913} C_VEL
LIN {X 0,Y 453.554,Z 527.989,A -85,B 0,C 180,E1 -8292.529,E2 -8292.529} C_VEL
LIN {X 0,Y 453.536,Z 527.99,A -85,B 0,C 180,E1 -8296.196,E2 -8296.196} C_VEL
LIN {X 0,Y 453.511,Z 527.991,A -85,B 0,C 180,E1 -8299.041,E2 -8299.041} C_VEL
LIN {X 0,Y 453.468,Z 527.995,A -85,B 0,C 180,E1 -8301.837,E2 -8301.837} C_VEL
LIN {X 0,Y 453.506,Z 527.996,A -85,B 0,C 180,E1 -8304.735,E2 -8304.735} C_VEL
LIN {X 0,Y 453.531,Z 527.985,A -85,B 0,C 180,E1 -8307.962,E2 -8307.962} C_VEL
LIN {X 0,Y 453.476,Z 528,A -85,B 0,C 180,E1 -8310.76,E2 -8310.76} C_VEL
LIN {X 0,Y 453.471,Z 527.996,A -85,B 0,C 180,E1 -8313.913,E2 -8313.913} C_VEL
LIN {X 0,Y 453.465,Z 527.997,A -85,B 0,C 180,E1 -8317.189,E2 -8317.189} C_VEL
LIN {X 0,Y 453.525,Z 527.988,A -85,B 0,C 180,E1 -8319.446,E2 -8319.446} C_VEL
LIN {X 0,Y 453.458,Z 528,A -85,B 0,C 180,E1 -8322.996,E2 -8322.996} C_VEL
LIN {X 0,Y 453.469,Z 527.996,A -85,B 0,C 180,E1 -8325.781,E2 -8325.781} C_VEL
LIN {X 0,Y 453.478,Z 527.999,A -85,B 0,C 180,E1 -8328.21,E2 -8328.21} C_VEL
LIN {X 0,Y 453.512,Z 527.996,A -85,B 0,C 180,E1 -8330.791,E2 -8330.791} C_VEL
LIN {X 0,Y 453.452,Z 528,A -85,B 0,C 180,E1 -8333.918,E2 -8333.918} C_VEL
LIN {X 0,Y 453.482,Z 527.997,A -85,B 0,C 180,E1 -8337.152,E2 -8337.152} C_VEL
LIN {X 0,Y 453.475,Z 528,A -85,B 0,C 180,E1 -8340.269,E2 -8340.269} C_VEL
LIN {X 0,Y 453.533,Z 527.993,A -85,B 0,C 180,E1 -8343.296,E2 -8343.296} C_VEL
LIN {X 0,Y 453.543,Z 528.1,A -85,B 0,C 180,E1 -8343.657,E2 -8343.657} C_VEL
LIN {X 0,Y 455.954,Z 540.244,A -85,B 0,C 180,E1 -8346.168,E2 -8346.168} C_VEL
LIN {X 0,Y 455.982,Z 545.08,A -85,B 0,C 180,E1 -8347.097,E2 -8347.097} C_VEL
LIN {X 0,Y 455.003,Z 562.904,A -85,B 0,C 180,E1 -8350.426,E2 -8350.426} C_VEL
LIN {X 0,Y 454.49,Z 573.454,A -85,B 0,C 180,E1 -8352.375,E2 -8352.375} C_VEL
LIN {X 0,Y 457.804,Z 594.643,A -85,B 0,C 180,E1 -8352.868,E2 -8352.868} C_VEL
LIN {X 0,Y 457.037,Z 682.196,A -85,B 0,C 180,E1 -8354.275,E2 -8354.275} C_VEL
LIN {X 0,Y 456.527,Z 696.026,A -85,B 0,C 180,E1 -8354.686,E2 -8354.686} C_VEL
LIN {X 0,Y 456.006,Z 708.931,A -85,B 0,C 180,E1 -8355.268,E2 -8355.268} C_VEL
LIN {X 0,Y 455.39,Z 721.473,A -85,B 0,C 180,E1 -8356.047,E2 -8356.047} C_VEL
LIN {X 0,Y 454.83,Z 732.574,A -85,B 0,C 180,E1 -8356.932,E2 -8356.932} C_VEL
LIN {X 0,Y 454.305,Z 742.747,A -85,B 0,C 180,E1 -8357.946,E2 -8357.946} C_VEL
LIN {X 0,Y 453.751,Z 751.86,A -85,B 0,C 180,E1 -8359.063,E2 -8359.063} C_VEL
LIN {X 0,Y 453.286,Z 760.753,A -85,B 0,C 180,E1 -8360.406,E2 -8360.406} C_VEL
LIN {X 0,Y 452.938,Z 767.909,A -85,B 0,C 180,E1 -8361.748,E2 -8361.748} C_VEL
LIN {X 0,Y 452.724,Z 772.746,A -85,B 0,C 180,E1 -8362.866,E2 -8362.866} C_VEL
LIN {X 0,Y 452.584,Z 777.448,A -85,B 0,C 180,E1 -8364.207,E2 -8364.207} C_VEL
LIN {X 0,Y 452.491,Z 781.041,A -85,B 0,C 180,E1 -8365.546,E2 -8365.546} C_VEL
LIN {X 0,Y 452.482,Z 782.893,A -85,B 0,C 180,E1 -8366.438,E2 -8366.438} C_VEL
LIN {X 0,Y 452.508,Z 784.282,A -85,B 0,C 180,E1 -8367.329,E2 -8367.329} C_VEL
LIN {X 0,Y 452.428,Z 785.877,A -85,B 0,C 180,E1 -8369.11,E2 -8369.11} C_VEL
LIN {X 0,Y 452.434,Z 786.086,A -85,B 0,C 180,E1 -8370,E2 -8370} C_VEL
LIN {X 0,Y 452.436,Z 785.251,A -85,B 0,C 180,E1 -8371.78,E2 -8371.78} C_VEL
LIN {X 0,Y 452.508,Z 784.253,A -85,B 0,C 180,E1 -8372.671,E2 -8372.671} C_VEL
LIN {X 0,Y 452.483,Z 782.846,A -85,B 0,C 180,E1 -8373.562,E2 -8373.562} C_VEL
LIN {X 0,Y 452.552,Z 779.899,A -85,B 0,C 180,E1 -8374.9,E2 -8374.9} C_VEL
LIN {X 0,Y 452.628,Z 775.286,A -85,B 0,C 180,E1 -8376.416,E2 -8376.416} C_VEL
LIN {X 0,Y 452.893,Z 768.746,A -85,B 0,C 180,E1 -8378.028,E2 -8378.028} C_VEL
LIN {X 0,Y 453.21,Z 761.809,A -85,B 0,C 180,E1 -8379.371,E2 -8379.371} C_VEL
LIN {X 0,Y 453.614,Z 753.112,A -85,B 0,C 180,E1 -8380.715,E2 -8380.715} C_VEL
LIN {X 0,Y 454.184,Z 744.201,A -85,B 0,C 180,E1 -8381.831,E2 -8381.831} C_VEL
LIN {X 0,Y 454.731,Z 733.339,A -85,B 0,C 180,E1 -8382.938,E2 -8382.938} C_VEL
LIN {X 0,Y 455.331,Z 722.083,A -85,B 0,C 180,E1 -8383.841,E2 -8383.841} C_VEL
LIN {X 0,Y 455.763,Z 711.594,A -85,B 0,C 180,E1 -8384.511,E2 -8384.511} C_VEL
LIN {X 0,Y 456.26,Z 699.007,A -85,B 0,C 180,E1 -8385.123,E2 -8385.123} C_VEL
LIN {X 0,Y 456.699,Z 686.836,A -85,B 0,C 180,E1 -8385.537,E2 -8385.537} C_VEL
LIN {X 0,Y 456.954,Z 673.206,A -85,B 0,C 180,E1 -8385.814,E2 -8385.814} C_VEL
LIN {X 0,Y 457.411,Z 592.699,A -85,B 0,C 180,E1 -8387.083,E2 -8387.083} C_VEL
LIN {X 0,Y 454.411,Z 573.575,A -85,B 0,C 180,E1 -8387.5,E2 -8387.5} C_VEL
LIN {X 0,Y 455.15,Z 556.834,A -85,B 0,C 180,E1 -8390.565,E2 -8390.565} C_VEL
LIN {X 0,Y 455.967,Z 541.583,A -85,B 0,C 180,E1 -8393.384,E2 -8393.384} C_VEL
LIN {X 0,Y 453.943,Z 530.007,A -85,B 0,C 180,E1 -8395.689,E2 -8395.689} C_VEL
LIN {X 0,Y 453.559,Z 527.99,A -85,B 0,C 180,E1 -8396.108,E2 -8396.108} C_VEL
LIN {X 0,Y 453.51,Z 527.993,A -85,B 0,C 180,E1 -8398.711,E2 -8398.711} C_VEL
LIN {X 0,Y 453.464,Z 527.999,A -85,B 0,C 180,E1 -8401.799,E2 -8401.799} C_VEL
LIN {X 0,Y 453.478,Z 527.995,A -85,B 0,C 180,E1 -8404.988,E2 -8404.988} C_VEL
LIN {X 0,Y 453.47,Z 527.994,A -85,B 0,C 180,E1 -8408.31,E2 -8408.31} C_VEL
LIN {X 0,Y 453.491,Z 527.992,A -85,B 0,C 180,E1 -8410.608,E2 -8410.608} C_VEL
LIN {X 0,Y 453.459,Z 528,A -85,B 0,C 180,E1 -8413.244,E2 -8413.244} C_VEL
LIN {X 0,Y 453.461,Z 527.999,A -85,B 0,C 180,E1 -8415.778,E2 -8415.778} C_VEL
LIN {X 0,Y 453.511,Z 527.997,A -85,B 0,C 180,E1 -8419.405,E2 -8419.405} C_VEL
LIN {X 0,Y 453.471,Z 527.994,A -85,B 0,C 180,E1 -8422.222,E2 -8422.222} C_VEL
LIN {X 0,Y 453.483,Z 527.997,A -85,B 0,C 180,E1 -8425.222,E2 -8425.222} C_VEL
LIN {X 0,Y 453.461,Z 527.995,A -85,B 0,C 180,E1 -8428.474,E2 -8428.474} C_VEL
LIN {X 0,Y 453.508,Z 527.995,A -85,B 0,C 180,E1 -8431.288,E2 -8431.288} C_VEL
LIN {X 0,Y 453.517,Z 527.988,A -85,B 0,C 180,E1 -8434.284,E2 -8434.284} C_VEL
LIN {X 0,Y 453.471,Z 527.999,A -85,B 0,C 180,E1 -8437.204,E2 -8437.204} C_VEL
LIN {X 0,Y 453.496,Z 527.992,A -85,B 0,C 180,E1 -8440.066,E2 -8440.066} C_VEL
LIN {X 0,Y 453.498,Z 527.992,A -85,B 0,C 180,E1 -8442.876,E2 -8442.876} C_VEL
LIN {X 0,Y 453.506,Z 527.995,A -85,B 0,C 180,E1 -8445.644,E2 -8445.644} C_VEL
LIN {X 0,Y 453.552,Z 527.984,A -85,B 0,C 180,E1 -8448.379,E2 -8448.379} C_VEL
LIN {X 0,Y 453.642,Z 527.974,A -85,B 0,C 180,E1 -8451.985,E2 -8451.985} C_VEL
LIN {X 0,Y 453.663,Z 527.97,A -85,B 0,C 180,E1 -8454.667,E2 -8454.667} C_VEL
LIN {X 0,Y 453.757,Z 527.965,A -85,B 0,C 180,E1 -8457.337,E2 -8457.337} C_VEL
LIN {X 0,Y 453.813,Z 527.953,A -85,B 0,C 180,E1 -8460,E2 -8460} C_VEL
LIN {X 0,Y 453.757,Z 527.959,A -85,B 0,C 180,E1 -8462.663,E2 -8462.663} C_VEL
LIN {X 0,Y 453.673,Z 527.969,A -85,B 0,C 180,E1 -8466.225,E2 -8466.225} C_VEL
LIN {X 0,Y 453.584,Z 527.982,A -85,B 0,C 180,E1 -8468.914,E2 -8468.914} C_VEL
LIN {X 0,Y 453.554,Z 527.984,A -85,B 0,C 180,E1 -8472.529,E2 -8472.529} C_VEL
LIN {X 0,Y 453.536,Z 527.986,A -85,B 0,C 180,E1 -8476.196,E2 -8476.196} C_VEL
LIN {X 0,Y 453.512,Z 527.992,A -85,B 0,C 180,E1 -8479.041,E2 -8479.041} C_VEL
LIN {X 0,Y 453.469,Z 527.997,A -85,B 0,C 180,E1 -8481.837,E2 -8481.837} C_VEL
LIN {X 0,Y 453.507,Z 527.99,A -85,B 0,C 180,E1 -8484.735,E2 -8484.735} C_VEL
LIN {X 0,Y 453.532,Z 527.988,A -85,B 0,C 180,E1 -8487.962,E2 -8487.962} C_VEL
LIN {X 0,Y 453.477,Z 527.994,A -85,B 0,C 180,E1 -8490.76,E2 -8490.76} C_VEL
LIN {X 0,Y 453.472,Z 527.996,A -85,B 0,C 180,E1 -8493.913,E2 -8493.913} C_VEL
LIN {X 0,Y 453.466,Z 528,A -85,B 0,C 180,E1 -8497.189,E2 -8497.189} C_VEL
LIN {X 0,Y 453.513,Z 527.997,A -85,B 0,C 180,E1 -8499.448,E2 -8499.448} C_VEL
LIN {X 0,Y 453.464,Z 527.998,A -85,B 0,C 180,E1 -8502.995,E2 -8502.995} C_VEL
LIN {X 0,Y 453.474,Z 527.997,A -85,B 0,C 180,E1 -8505.781,E2 -8505.781} C_VEL
LIN {X 0,Y 453.494,Z 527.991,A -85,B 0,C 180,E1 -8508.212,E2 -8508.212} C_VEL
LIN {X 0,Y 453.529,Z 527.988,A -85,B 0,C 180,E1 -8510.789,E2 -8510.789} C_VEL
LIN {X 0,Y 453.455,Z 527.998,A -85,B 0,C 180,E1 -8513.918,E2 -8513.918} C_VEL
LIN {X 0,Y 453.483,Z 527.997,A -85,B 0,C 180,E1 -8517.152,E2 -8517.152} C_VEL
LIN {X 0,Y 453.475,Z 527.993,A -85,B 0,C 180,E1 -8520.269,E2 -8520.269} C_VEL
LIN {X 0,Y 453.508,Z 527.996,A -85,B 0,C 180,E1 -8523.295,E2 -8523.295} C_VEL
LIN {X 0,Y 453.505,Z 527.99,A -85,B 0,C 180,E1 -8526.24,E2 -8526.24} C_VEL
LIN {X 0,Y 453.486,Z 528.002,A -85,B 0,C 180,E1 -8529.118,E2 -8529.118} C_VEL
LIN {X 0,Y 453.581,Z 528.093,A -85,B 0,C 180,E1 -8531.773,E2 -8531.773} C_VEL
LIN {X 0,Y 454.935,Z 535.481,A -85,B 0,C 180,E1 -8533.499,E2 -8533.499} C_VEL
LIN {X 0,Y 454.789,Z 543.321,A -85,B 0,C 180,E1 -8535.228,E2 -8535.228} C_VEL
LIN {X 0,Y 454.549,Z 549.688,A -85,B 0,C 180,E1 -8536.576,E2 -8536.576} C_VEL
LIN {X 0,Y 457.603,Z 565.401,A -85,B 0,C 180,E1 -8536.942,E2 -8536.942} C_VEL
LIN {X 0,Y 457.512,Z 594.139,A -85,B 0,C 180,E1 -8537.398,E2 -8537.398} C_VEL
LIN {X 0,Y 456.892,Z 599.981,A -85,B 0,C 180,E1 -8537.47,E2 -8537.47} C_VEL
LIN {X 0,Y 451.193,Z 618.976,A -85,B 0,C 180,E1 -8537.574,E2 -8537.574} C_VEL
LIN {X 0,Y 450.439,Z 624.824,A -85,B 0,C 180,E1 -8537.642,E2 -8537.642} C_VEL
LIN {X 0,Y 450.064,Z 656.865,A -85,B 0,C 180,E1 -8538.173,E2 -8538.173} C_VEL
LIN {X 0,Y 449.716,Z 669.914,A -85,B 0,C 180,E1 -8538.564,E2 -8538.564} C_VEL
LIN {X 0,Y 449.315,Z 682.483,A -85,B 0,C 180,E1 -8539.125,E2 -8539.125} C_VEL
LIN {X 0,Y 448.788,Z 694.468,A -85,B 0,C 180,E1 -8539.853,E2 -8539.853} C_VEL
LIN {X 0,Y 448.224,Z 705.876,A -85,B 0,C 180,E1 -8540.752,E2 -8540.752} C_VEL
LIN {X 0,Y 447.532,Z 715.324,A -85,B 0,C 180,E1 -8541.67,E2 -8541.67} C_VEL
LIN {X 0,Y 447.163,Z 723.049,A -85,B 0,C 180,E1 -8542.58,E2 -8542.58} C_VEL
LIN {X 0,Y 446.767,Z 732.332,A -85,B 0,C 180,E1 -8543.905,E2 -8543.905} C_VEL
LIN {X 0,Y 446.277,Z 739.927,A -85,B 0,C 180,E1 -8545.258,E2 -8545.258} C_VEL
LIN {X 0,Y 445.891,Z 746.928,A -85,B 0,C 180,E1 -8546.838,E2 -8546.838} C_VEL
LIN {X 0,Y 445.543,Z 751.596,A -85,B 0,C 180,E1 -8548.192,E2 -8548.192} C_VEL
LIN {X 0,Y 445.474,Z 755.162,A -85,B 0,C 180,E1 -8549.548,E2 -8549.548} C_VEL
LIN {X 0,Y 445.369,Z 757.735,A -85,B 0,C 180,E1 -8550.904,E2 -8550.904} C_VEL
LIN {X 0,Y 445.379,Z 758.947,A -85,B 0,C 180,E1 -8551.808,E2 -8551.808} C_VEL
LIN {X 0,Y 445.439,Z 759.738,A -85,B 0,C 180,E1 -8552.713,E2 -8552.713} C_VEL
LIN {X 0,Y 445.352,Z 760.129,A -85,B 0,C 180,E1 -8554.525,E2 -8554.525} C_VEL
LIN {X 0,Y 445.433,Z 759.047,A -85,B 0,C 180,E1 -8556.272,E2 -8556.272} C_VEL
LIN {X 0,Y 445.457,Z 757.754,A -85,B 0,C 180,E1 -8557.251,E2 -8557.251} C_VEL
LIN {X 0,Y 445.519,Z 755.174,A -85,B 0,C 180,E1 -8558.619,E2 -8558.619} C_VEL
LIN {X 0,Y 445.605,Z 751.578,A -85,B 0,C 180,E1 -8559.991,E2 -8559.991} C_VEL
LIN {X 0,Y 445.926,Z 746.855,A -85,B 0,C 180,E1 -8561.362,E2 -8561.362} C_VEL
LIN {X 0,Y 446.204,Z 740.862,A -85,B 0,C 180,E1 -8562.739,E2 -8562.739} C_VEL
LIN {X 0,Y 446.66,Z 733.38,A -85,B 0,C 180,E1 -8564.116,E2 -8564.116} C_VEL
LIN {X 0,Y 447.124,Z 725.722,A -85,B 0,C 180,E1 -8565.264,E2 -8565.264} C_VEL
LIN {X 0,Y 447.727,Z 716.392,A -85,B 0,C 180,E1 -8566.412,E2 -8566.412} C_VEL
LIN {X 0,Y 448.256,Z 705.96,A -85,B 0,C 180,E1 -8567.448,E2 -8567.448} C_VEL
LIN {X 0,Y 448.951,Z 694.354,A -85,B 0,C 180,E1 -8568.363,E2 -8568.363} C_VEL
LIN {X 0,Y 449.559,Z 682.062,A -85,B 0,C 180,E1 -8569.106,E2 -8569.106} C_VEL
LIN {X 0,Y 449.972,Z 669.044,A -85,B 0,C 180,E1 -8569.68,E2 -8569.68} C_VEL
LIN {X 0,Y 450.328,Z 656.402,A -85,B 0,C 180,E1 -8570.05,E2 -8570.05} C_VEL
LIN {X 0,Y 451.112,Z 566.529,A -85,B 0,C 180,E1 -8571.514,E2 -8571.514} C_VEL
LIN {X 0,Y 447.731,Z 549.694,A -85,B 0,C 180,E1 -8571.964,E2 -8571.964} C_VEL
LIN {X 0,Y 448.204,Z 538.729,A -85,B 0,C 180,E1 -8574.419,E2 -8574.419} C_VEL
LIN {X 0,Y 446.904,Z 530.869,A -85,B 0,C 180,E1 -8576.313,E2 -8576.313} C_VEL
LIN {X 0,Y 446.503,Z 528.869,A -85,B 0,C 180,E1 -8576.858,E2 -8576.858} C_VEL
LIN {X 0,Y 446.428,Z 528.874,A -85,B 0,C 180,E1 -8580.249,E2 -8580.249} C_VEL
LIN {X 0,Y 446.445,Z 528.873,A -85,B 0,C 180,E1 -8583.453,E2 -8583.453} C_VEL
LIN {X 0,Y 446.408,Z 528.882,A -85,B 0,C 180,E1 -8586.744,E2 -8586.744} C_VEL
LIN {X 0,Y 446.49,Z 528.866,A -85,B 0,C 180,E1 -8589.53,E2 -8589.53} C_VEL
LIN {X 0,Y 446.448,Z 528.876,A -85,B 0,C 180,E1 -8592.601,E2 -8592.601} C_VEL
LIN {X 0,Y 446.454,Z 528.871,A -85,B 0,C 180,E1 -8595.102,E2 -8595.102} C_VEL
LIN {X 0,Y 446.431,Z 528.871,A -85,B 0,C 180,E1 -8598.609,E2 -8598.609} C_VEL
LIN {X 0,Y 446.46,Z 528.873,A -85,B 0,C 180,E1 -8600.974,E2 -8600.974} C_VEL
LIN {X 0,Y 446.416,Z 528.877,A -85,B 0,C 180,E1 -8604.373,E2 -8604.373} C_VEL
LIN {X 0,Y 446.417,Z 528.874,A -85,B 0,C 180,E1 -8607.638,E2 -8607.638} C_VEL
LIN {X 0,Y 446.463,Z 528.874,A -85,B 0,C 180,E1 -8610.791,E2 -8610.791} C_VEL
LIN {X 0,Y 446.471,Z 528.864,A -85,B 0,C 180,E1 -8613.848,E2 -8613.848} C_VEL
LIN {X 0,Y 446.421,Z 528.874,A -85,B 0,C 180,E1 -8616.823,E2 -8616.823} C_VEL
LIN {X 0,Y 446.436,Z 528.871,A -85,B 0,C 180,E1 -8619.737,E2 -8619.737} C_VEL
LIN {X 0,Y 446.455,Z 528.871,A -85,B 0,C 180,E1 -8622.597,E2 -8622.597} C_VEL
LIN {X 0,Y 446.461,Z 528.868,A -85,B 0,C 180,E1 -8625.412,E2 -8625.412} C_VEL
LIN {X 0,Y 446.51,Z 528.86,A -85,B 0,C 180,E1 -8628.193,E2 -8628.193} C_VEL
LIN {X 0,Y 446.591,Z 528.849,A -85,B 0,C 180,E1 -8631.857,E2 -8631.857} C_VEL
LIN {X 0,Y 446.64,Z 528.852,A -85,B 0,C 180,E1 -8634.582,E2 -8634.582} C_VEL
LIN {X 0,Y 446.701,Z 528.834,A -85,B 0,C 180,E1 -8637.295,E2 -8637.295} C_VEL
LIN {X 0,Y 446.785,Z 528.828,A -85,B 0,C 180,E1 -8640,E2 -8640} C_VEL
LIN {X 0,Y 446.701,Z 528.839,A -85,B 0,C 180,E1 -8642.705,E2 -8642.705} C_VEL
LIN {X 0,Y 446.637,Z 528.85,A -85,B 0,C 180,E1 -8646.324,E2 -8646.324} C_VEL
LIN {X 0,Y 446.53,Z 528.86,A -85,B 0,C 180,E1 -8649.055,E2 -8649.055} C_VEL
LIN {X 0,Y 446.512,Z 528.862,A -85,B 0,C 180,E1 -8652.73,E2 -8652.73} C_VEL
LIN {X 0,Y 446.487,Z 528.868,A -85,B 0,C 180,E1 -8656.228,E2 -8656.228} C_VEL
LIN {X 0,Y 446.461,Z 528.868,A -85,B 0,C 180,E1 -8659.304,E2 -8659.304} C_VEL
LIN {X 0,Y 446.41,Z 528.877,A -85,B 0,C 180,E1 -8662.2,E2 -8662.2} C_VEL
LIN {X 0,Y 446.45,Z 528.871,A -85,B 0,C 180,E1 -8665.153,E2 -8665.153} C_VEL
LIN {X 0,Y 446.477,Z 528.865,A -85,B 0,C 180,E1 -8668.179,E2 -8668.179} C_VEL
LIN {X 0,Y 446.413,Z 528.875,A -85,B 0,C 180,E1 -8671.301,E2 -8671.301} C_VEL
LIN {X 0,Y 446.424,Z 528.879,A -85,B 0,C 180,E1 -8674.523,E2 -8674.523} C_VEL
LIN {X 0,Y 446.431,Z 528.874,A -85,B 0,C 180,E1 -8678.084,E2 -8678.084} C_VEL
LIN {X 0,Y 446.438,Z 528.875,A -85,B 0,C 180,E1 -8680.921,E2 -8680.921} C_VEL
LIN {X 0,Y 446.397,Z 528.878,A -85,B 0,C 180,E1 -8683.847,E2 -8683.847} C_VEL
LIN {X 0,Y 446.417,Z 528.88,A -85,B 0,C 180,E1 -8686.401,E2 -8686.401} C_VEL
LIN {X 0,Y 446.448,Z 528.871,A -85,B 0,C 180,E1 -8689.804,E2 -8689.804} C_VEL
LIN {X 0,Y 446.425,Z 528.877,A -85,B 0,C 180,E1 -8692.124,E2 -8692.124} C_VEL
LIN {X 0,Y 446.427,Z 528.874,A -85,B 0,C 180,E1 -8695.478,E2 -8695.478} C_VEL
LIN {X 0,Y 446.415,Z 528.879,A -85,B 0,C 180,E1 -8698.7,E2 -8698.7} C_VEL
LIN {X 0,Y 446.484,Z 528.869,A -85,B 0,C 180,E1 -8701.822,E2 -8701.822} C_VEL
LIN {X 0,Y 446.527,Z 529.042,A -85,B 0,C 180,E1 -8703.41,E2 -8703.41} C_VEL
LIN {X 0,Y 448.957,Z 541.253,A -85,B 0,C 180,E1 -8705.984,E2 -8705.984} C_VEL
LIN {X 0,Y 449.168,Z 545.012,A -85,B 0,C 180,E1 -8706.73,E2 -8706.73} C_VEL
LIN {X 0,Y 448.16,Z 561.272,A -85,B 0,C 180,E1 -8709.819,E2 -8709.819} C_VEL
LIN {X 0,Y 447.566,Z 573.278,A -85,B 0,C 180,E1 -8712.08,E2 -8712.08} C_VEL
LIN {X 0,Y 451.044,Z 594.737,A -85,B 0,C 180,E1 -8712.59,E2 -8712.59} C_VEL
LIN {X 0,Y 450.242,Z 681.527,A -85,B 0,C 180,E1 -8714.002,E2 -8714.002} C_VEL
LIN {X 0,Y 449.756,Z 694.747,A -85,B 0,C 180,E1 -8714.392,E2 -8714.392} C_VEL
LIN {X 0,Y 449.252,Z 707.994,A -85,B 0,C 180,E1 -8714.984,E2 -8714.984} C_VEL
LIN {X 0,Y 448.593,Z 719.915,A -85,B 0,C 180,E1 -8715.715,E2 -8715.715} C_VEL
LIN {X 0,Y 447.969,Z 730.898,A -85,B 0,C 180,E1 -8716.58,E2 -8716.58} C_VEL
LIN {X 0,Y 447.423,Z 741.67,A -85,B 0,C 180,E1 -8717.642,E2 -8717.642} C_VEL
LIN {X 0,Y 446.852,Z 750.115,A -85,B 0,C 180,E1 -8718.662,E2 -8718.662} C_VEL
LIN {X 0,Y 446.33,Z 759.278,A -85,B 0,C 180,E1 -8720.026,E2 -8720.026} C_VEL
LIN {X 0,Y 445.935,Z 766.663,A -85,B 0,C 180,E1 -8721.389,E2 -8721.389} C_VEL
LIN {X 0,Y 445.669,Z 772.597,A -85,B 0,C 180,E1 -8722.753,E2 -8722.753} C_VEL
LIN {X 0,Y 445.495,Z 776.688,A -85,B 0,C 180,E1 -8723.925,E2 -8723.925} C_VEL
LIN {X 0,Y 445.417,Z 780.867,A -85,B 0,C 180,E1 -8725.475,E2 -8725.475} C_VEL
LIN {X 0,Y 445.381,Z 782.71,A -85,B 0,C 180,E1 -8726.381,E2 -8726.381} C_VEL
LIN {X 0,Y 445.433,Z 784.094,A -85,B 0,C 180,E1 -8727.287,E2 -8727.287} C_VEL
LIN {X 0,Y 445.338,Z 785.679,A -85,B 0,C 180,E1 -8729.096,E2 -8729.096} C_VEL
LIN {X 0,Y 445.342,Z 785.881,A -85,B 0,C 180,E1 -8730,E2 -8730} C_VEL
LIN {X 0,Y 445.355,Z 785.036,A -85,B 0,C 180,E1 -8731.809,E2 -8731.809} C_VEL
LIN {X 0,Y 445.433,Z 784.033,A -85,B 0,C 180,E1 -8732.713,E2 -8732.713} C_VEL
LIN {X 0,Y 445.382,Z 782.617,A -85,B 0,C 180,E1 -8733.619,E2 -8733.619} C_VEL
LIN {X 0,Y 445.481,Z 779.662,A -85,B 0,C 180,E1 -8734.978,E2 -8734.978} C_VEL
LIN {X 0,Y 445.576,Z 774.21,A -85,B 0,C 180,E1 -8736.748,E2 -8736.748} C_VEL
LIN {X 0,Y 445.846,Z 768.479,A -85,B 0,C 180,E1 -8738.156,E2 -8738.156} C_VEL
LIN {X 0,Y 446.159,Z 761.523,A -85,B 0,C 180,E1 -8739.52,E2 -8739.52} C_VEL
LIN {X 0,Y 446.6,Z 752.798,A -85,B 0,C 180,E1 -8740.885,E2 -8740.885} C_VEL
LIN {X 0,Y 447.216,Z 743.865,A -85,B 0,C 180,E1 -8742.018,E2 -8742.018} C_VEL
LIN {X 0,Y 447.748,Z 733.657,A -85,B 0,C 180,E1 -8743.077,E2 -8743.077} C_VEL
LIN {X 0,Y 448.325,Z 723.244,A -85,B 0,C 180,E1 -8743.946,E2 -8743.946} C_VEL
LIN {X 0,Y 448.883,Z 711.108,A -85,B 0,C 180,E1 -8744.739,E2 -8744.739} C_VEL
LIN {X 0,Y 449.4,Z 698.427,A -85,B 0,C 180,E1 -8745.359,E2 -8745.359} C_VEL
LIN {X 0,Y 449.861,Z 686.015,A -85,B 0,C 180,E1 -8745.779,E2 -8745.779} C_VEL
LIN {X 0,Y 450.124,Z 670.161,A -85,B 0,C 180,E1 -8746.089,E2 -8746.089} C_VEL
LIN {X 0,Y 450.661,Z 593.942,A -85,B 0,C 180,E1 -8747.306,E2 -8747.306} C_VEL
LIN {X 0,Y 447.445,Z 573.239,A -85,B 0,C 180,E1 -8747.788,E2 -8747.788} C_VEL
LIN {X 0,Y 448.353,Z 555.269,A -85,B 0,C 180,E1 -8751.132,E2 -8751.132} C_VEL
LIN {X 0,Y 449.005,Z 542.562,A -85,B 0,C 180,E1 -8753.524,E2 -8753.524} C_VEL
LIN {X 0,Y 446.672,Z 529.698,A -85,B 0,C 180,E1 -8756.139,E2 -8756.139} C_VEL
LIN {X 0,Y 446.506,Z 528.867,A -85,B 0,C 180,E1 -8756.375,E2 -8756.375} C_VEL
LIN {X 0,Y 446.449,Z 528.876,A -85,B 0,C 180,E1 -8759.209,E2 -8759.209} C_VEL
LIN {X 0,Y 446.421,Z 528.872,A -85,B 0,C 180,E1 -8762.361,E2 -8762.361} C_VEL
LIN {X 0,Y 446.417,Z 528.879,A -85,B 0,C 180,E1 -8765.625,E2 -8765.625} C_VEL
LIN {X 0,Y 446.458,Z 528.87,A -85,B 0,C 180,E1 -8769.024,E2 -8769.024} C_VEL
LIN {X 0,Y 446.428,Z 528.871,A -85,B 0,C 180,E1 -8772.603,E2 -8772.603} C_VEL
LIN {X 0,Y 446.45,Z 528.872,A -85,B 0,C 180,E1 -8775.103,E2 -8775.103} C_VEL
LIN {X 0,Y 446.43,Z 528.871,A -85,B 0,C 180,E1 -8778.609,E2 -8778.609} C_VEL
LIN {X 0,Y 446.468,Z 528.869,A -85,B 0,C 180,E1 -8780.975,E2 -8780.975} C_VEL
LIN {X 0,Y 446.415,Z 528.873,A -85,B 0,C 180,E1 -8784.373,E2 -8784.373} C_VEL
LIN {X 0,Y 446.416,Z 528.878,A -85,B 0,C 180,E1 -8787.638,E2 -8787.638} C_VEL
LIN {X 0,Y 446.462,Z 528.868,A -85,B 0,C 180,E1 -8790.792,E2 -8790.792} C_VEL
LIN {X 0,Y 446.47,Z 528.869,A -85,B 0,C 180,E1 -8793.848,E2 -8793.848} C_VEL
LIN {X 0,Y 446.42,Z 528.873,A -85,B 0,C 180,E1 -8796.823,E2 -8796.823} C_VEL
LIN {X 0,Y 446.436,Z 528.875,A -85,B 0,C 180,E1 -8799.737,E2 -8799.737} C_VEL
LIN {X 0,Y 446.455,Z 528.868,A -85,B 0,C 180,E1 -8802.597,E2 -8802.597} C_VEL
LIN {X 0,Y 446.462,Z 528.875,A -85,B 0,C 180,E1 -8805.412,E2 -8805.412} C_VEL
LIN {X 0,Y 446.509,Z 528.862,A -85,B 0,C 180,E1 -8808.193,E2 -8808.193} C_VEL
LIN {X 0,Y 446.591,Z 528.854,A -85,B 0,C 180,E1 -8811.858,E2 -8811.858} C_VEL
LIN {X 0,Y 446.637,Z 528.845,A -85,B 0,C 180,E1 -8814.583,E2 -8814.583} C_VEL
LIN {X 0,Y 446.701,Z 528.844,A -85,B 0,C 180,E1 -8817.295,E2 -8817.295} C_VEL
LIN {X 0,Y 446.784,Z 528.829,A -85,B 0,C 180,E1 -8820,E2 -8820} C_VEL
LIN {X 0,Y 446.701,Z 528.838,A -85,B 0,C 180,E1 -8822.705,E2 -8822.705} C_VEL
LIN {X 0,Y 446.642,Z 528.845,A -85,B 0,C 180,E1 -8826.324,E2 -8826.324} C_VEL
LIN {X 0,Y 446.53,Z 528.862,A -85,B 0,C 180,E1 -8829.056,E2 -8829.056} C_VEL
LIN {X 0,Y 446.513,Z 528.862,A -85,B 0,C 180,E1 -8832.73,E2 -8832.73} C_VEL
LIN {X 0,Y 446.488,Z 528.864,A -85,B 0,C 180,E1 -8836.228,E2 -8836.228} C_VEL
LIN {X 0,Y 446.461,Z 528.874,A -85,B 0,C 180,E1 -8839.304,E2 -8839.304} C_VEL
LIN {X 0,Y 446.41,Z 528.874,A -85,B 0,C 180,E1 -8842.2,E2 -8842.2} C_VEL
LIN {X 0,Y 446.451,Z 528.873,A -85,B 0,C 180,E1 -8845.153,E2 -8845.153} C_VEL
LIN {X 0,Y 446.478,Z 528.866,A -85,B 0,C 180,E1 -8848.179,E2 -8848.179} C_VEL
LIN {X 0,Y 446.425,Z 528.878,A -85,B 0,C 180,E1 -8851.3,E2 -8851.3} C_VEL
LIN {X 0,Y 446.425,Z 528.872,A -85,B 0,C 180,E1 -8854.524,E2 -8854.524} C_VEL
LIN {X 0,Y 446.426,Z 528.872,A -85,B 0,C 180,E1 -8858.083,E2 -8858.083} C_VEL
LIN {X 0,Y 446.424,Z 528.874,A -85,B 0,C 180,E1 -8860.919,E2 -8860.919} C_VEL
LIN {X 0,Y 446.419,Z 528.875,A -85,B 0,C 180,E1 -8863.844,E2 -8863.844} C_VEL
LIN {X 0,Y 446.444,Z 528.869,A -85,B 0,C 180,E1 -8866.398,E2 -8866.398} C_VEL
LIN {X 0,Y 446.467,Z 528.869,A -85,B 0,C 180,E1 -8869.806,E2 -8869.806} C_VEL
LIN {X 0,Y 446.431,Z 528.871,A -85,B 0,C 180,E1 -8872.125,E2 -8872.125} C_VEL
LIN {X 0,Y 446.43,Z 528.878,A -85,B 0,C 180,E1 -8875.478,E2 -8875.478} C_VEL
LIN {X 0,Y 446.416,Z 528.874,A -85,B 0,C 180,E1 -8878.701,E2 -8878.701} C_VEL
LIN {X 0,Y 446.485,Z 528.867,A -85,B 0,C 180,E1 -8881.822,E2 -8881.822} C_VEL
LIN {X 0,Y 446.459,Z 528.869,A -85,B 0,C 180,E1 -8884.848,E2 -8884.848} C_VEL
LIN {X 0,Y 446.45,Z 528.873,A -85,B 0,C 180,E1 -8888.246,E2 -8888.246} C_VEL
LIN {X 0,Y 446.546,Z 529.01,A -85,B 0,C 180,E1 -8891.598,E2 -8891.598} C_VEL
LIN {X 0,Y 447.996,Z 537.477,A -85,B 0,C 180,E1 -8893.598,E2 -8893.598} C_VEL
LIN {X 0,Y 447.657,Z 547.924,A -85,B 0,C 180,E1 -8895.916,E2 -8895.916} C_VEL
LIN {X 0,Y 447.583,Z 549.697,A -85,B 0,C 180,E1 -8896.305,E2 -8896.305} C_VEL
LIN {X 0,Y 450.853,Z 566.711,A -85,B 0,C 180,E1 -8896.713,E2 -8896.713} C_VEL
LIN {X 0,Y 450.439,Z 624.824,A -85,B 0,C 180,E1 -8897.642,E2 -8897.642} C_VEL
LIN {X 0,Y 449.706,Z 630.667,A -85,B 0,C 180,E1 -8897.708,E2 -8897.708} C_VEL
LIN {X 0,Y 444.013,Z 649.642,A -85,B 0,C 180,E1 -8897.813,E2 -8897.813} C_VEL
LIN {X 0,Y 443.257,Z 655.456,A -85,B 0,C 180,E1 -8897.905,E2 -8897.905} C_VEL
LIN {X 0,Y 442.921,Z 668.333,A -85,B 0,C 180,E1 -8898.27,E2 -8898.27} C_VEL
LIN {X 0,Y 442.467,Z 681.37,A -85,B 0,C 180,E1 -8898.838,E2 -8898.838} C_VEL
LIN {X 0,Y 441.943,Z 693.741,A -85,B 0,C 180,E1 -8899.579,E2 -8899.579} C_VEL
LIN {X 0,Y 441.35,Z 705.328,A -85,B 0,C 180,E1 -8900.491,E2 -8900.491} C_VEL
LIN {X 0,Y 440.499,Z 716.71,A -85,B 0,C 180,E1 -8901.617,E2 -8901.617} C_VEL
LIN {X 0,Y 440.01,Z 725.15,A -85,B 0,C 180,E1 -8902.659,E2 -8902.659} C_VEL
LIN {X 0,Y 439.75,Z 732.831,A -85,B 0,C 180,E1 -8903.807,E2 -8903.807} C_VEL
LIN {X 0,Y 439.229,Z 740.364,A -85,B 0,C 180,E1 -8905.181,E2 -8905.181} C_VEL
LIN {X 0,Y 438.836,Z 747.321,A -85,B 0,C 180,E1 -8906.787,E2 -8906.787} C_VEL
LIN {X 0,Y 438.459,Z 751.951,A -85,B 0,C 180,E1 -8908.163,E2 -8908.163} C_VEL
LIN {X 0,Y 438.401,Z 755.478,A -85,B 0,C 180,E1 -8909.541,E2 -8909.541} C_VEL
LIN {X 0,Y 438.281,Z 758.016,A -85,B 0,C 180,E1 -8910.919,E2 -8910.919} C_VEL
LIN {X 0,Y 438.299,Z 759.209,A -85,B 0,C 180,E1 -8911.838,E2 -8911.838} C_VEL
LIN {X 0,Y 438.363,Z 759.968,A -85,B 0,C 180,E1 -8912.757,E2 -8912.757} C_VEL
LIN {X 0,Y 438.276,Z 760.325,A -85,B 0,C 180,E1 -8914.599,E2 -8914.599} C_VEL
LIN {X 0,Y 438.337,Z 759.33,A -85,B 0,C 180,E1 -8916.242,E2 -8916.242} C_VEL
LIN {X 0,Y 438.364,Z 757.883,A -85,B 0,C 180,E1 -8917.369,E2 -8917.369} C_VEL
LIN {X 0,Y 438.435,Z 755.267,A -85,B 0,C 180,E1 -8918.759,E2 -8918.759} C_VEL
LIN {X 0,Y 438.552,Z 751.632,A -85,B 0,C 180,E1 -8920.153,E2 -8920.153} C_VEL
LIN {X 0,Y 438.894,Z 746.87,A -85,B 0,C 180,E1 -8921.546,E2 -8921.546} C_VEL
LIN {X 0,Y 439.221,Z 740.833,A -85,B 0,C 180,E1 -8922.945,E2 -8922.945} C_VEL
LIN {X 0,Y 439.683,Z 733.302,A -85,B 0,C 180,E1 -8924.344,E2 -8924.344} C_VEL
LIN {X 0,Y 440.213,Z 725.588,A -85,B 0,C 180,E1 -8925.51,E2 -8925.51} C_VEL
LIN {X 0,Y 440.848,Z 716.152,A -85,B 0,C 180,E1 -8926.675,E2 -8926.675} C_VEL
LIN {X 0,Y 441.452,Z 705.632,A -85,B 0,C 180,E1 -8927.726,E2 -8927.726} C_VEL
LIN {X 0,Y 442.162,Z 693.903,A -85,B 0,C 180,E1 -8928.655,E2 -8928.655} C_VEL
LIN {X 0,Y 442.745,Z 682.476,A -85,B 0,C 180,E1 -8929.351,E2 -8929.351} C_VEL
LIN {X 0,Y 443.187,Z 669.537,A -85,B 0,C 180,E1 -8929.934,E2 -8929.934} C_VEL
LIN {X 0,Y 443.551,Z 657.041,A -85,B 0,C 180,E1 -8930.31,E2 -8930.31} C_VEL
LIN {X 0,Y 444.352,Z 567.193,A -85,B 0,C 180,E1 -8931.801,E2 -8931.801} C_VEL
LIN {X 0,Y 440.83,Z 549.952,A -85,B 0,C 180,E1 -8932.264,E2 -8932.264} C_VEL
LIN {X 0,Y 441.284,Z 540.269,A -85,B 0,C 180,E1 -8934.461,E2 -8934.461} C_VEL
LIN {X 0,Y 439.878,Z 531.826,A -85,B 0,C 180,E1 -8936.527,E2 -8936.527} C_VEL
LIN {X 0,Y 439.481,Z 529.745,A -85,B 0,C 180,E1 -8937.049,E2 -8937.049} C_VEL
LIN {X 0,Y 439.381,Z 529.751,A -85,B 0,C 180,E1 -8940.26,E2 -8940.26} C_VEL
LIN {X 0,Y 439.396,Z 529.751,A -85,B 0,C 180,E1 -8943.723,E2 -8943.723} C_VEL
LIN {X 0,Y 439.357,Z 529.758,A -85,B 0,C 180,E1 -8946.888,E2 -8946.888} C_VEL
LIN {X 0,Y 439.426,Z 529.746,A -85,B 0,C 180,E1 -8949.852,E2 -8949.852} C_VEL
LIN {X 0,Y 439.401,Z 529.755,A -85,B 0,C 180,E1 -8952.629,E2 -8952.629} C_VEL
LIN {X 0,Y 439.403,Z 529.748,A -85,B 0,C 180,E1 -8955.271,E2 -8955.271} C_VEL
LIN {X 0,Y 439.394,Z 529.746,A -85,B 0,C 180,E1 -8958.741,E2 -8958.741} C_VEL
LIN {X 0,Y 439.382,Z 529.75,A -85,B 0,C 180,E1 -8961.605,E2 -8961.605} C_VEL
LIN {X 0,Y 439.396,Z 529.753,A -85,B 0,C 180,E1 -8964.843,E2 -8964.843} C_VEL
LIN {X 0,Y 439.37,Z 529.754,A -85,B 0,C 180,E1 -8968.139,E2 -8968.139} C_VEL
LIN {X 0,Y 439.419,Z 529.746,A -85,B 0,C 180,E1 -8971.326,E2 -8971.326} C_VEL
LIN {X 0,Y 439.399,Z 529.749,A -85,B 0,C 180,E1 -8974.414,E2 -8974.414} C_VEL
LIN {X 0,Y 439.357,Z 529.749,A -85,B 0,C 180,E1 -8977.424,E2 -8977.424} C_VEL
LIN {X 0,Y 439.433,Z 529.749,A -85,B 0,C 180,E1 -8980.662,E2 -8980.662} C_VEL
LIN {X 0,Y 439.454,Z 529.743,A -85,B 0,C 180,E1 -8984.224,E2 -8984.224} C_VEL
LIN {X 0,Y 439.475,Z 529.735,A -85,B 0,C 180,E1 -8988.001,E2 -8988.001} C_VEL
LIN {X 0,Y 439.539,Z 529.727,A -85,B 0,C 180,E1 -8991.726,E2 -8991.726} C_VEL
LIN {X 0,Y 439.615,Z 529.725,A -85,B 0,C 180,E1 -8994.496,E2 -8994.496} C_VEL
LIN {X 0,Y 439.627,Z 529.716,A -85,B 0,C 180,E1 -8998.168,E2 -8998.168} C_VEL
LIN {X 0,Y 439.755,Z 529.704,A -85,B 0,C 180,E1 -9000,E2 -9000} C_VEL
LIN {X 0,Y 439.648,Z 529.716,A -85,B 0,C 180,E1 -9002.749,E2 -9002.749} C_VEL
LIN {X 0,Y 439.609,Z 529.727,A -85,B 0,C 180,E1 -9006.425,E2 -9006.425} C_VEL
LIN {X 0,Y 439.492,Z 529.735,A -85,B 0,C 180,E1 -9009.202,E2 -9009.202} C_VEL
LIN {X 0,Y 439.457,Z 529.739,A -85,B 0,C 180,E1 -9012.938,E2 -9012.938} C_VEL
LIN {X 0,Y 439.438,Z 529.747,A -85,B 0,C 180,E1 -9016.349,E2 -9016.349} C_VEL
LIN {X 0,Y 439.394,Z 529.747,A -85,B 0,C 180,E1 -9019.627,E2 -9019.627} C_VEL
LIN {X 0,Y 439.357,Z 529.755,A -85,B 0,C 180,E1 -9022.576,E2 -9022.576} C_VEL
LIN {X 0,Y 439.397,Z 529.748,A -85,B 0,C 180,E1 -9025.585,E2 -9025.585} C_VEL
LIN {X 0,Y 439.418,Z 529.752,A -85,B 0,C 180,E1 -9028.673,E2 -9028.673} C_VEL
LIN {X 0,Y 439.368,Z 529.752,A -85,B 0,C 180,E1 -9031.861,E2 -9031.861} C_VEL
LIN {X 0,Y 439.395,Z 529.75,A -85,B 0,C 180,E1 -9035.156,E2 -9035.156} C_VEL
LIN {X 0,Y 439.392,Z 529.756,A -85,B 0,C 180,E1 -9038.594,E2 -9038.594} C_VEL
LIN {X 0,Y 439.393,Z 529.75,A -85,B 0,C 180,E1 -9041.259,E2 -9041.259} C_VEL
LIN {X 0,Y 439.398,Z 529.754,A -85,B 0,C 180,E1 -9044.73,E2 -9044.73} C_VEL
LIN {X 0,Y 439.394,Z 529.75,A -85,B 0,C 180,E1 -9047.797,E2 -9047.797} C_VEL
LIN {X 0,Y 439.434,Z 529.748,A -85,B 0,C 180,E1 -9050.229,E2 -9050.229} C_VEL
LIN {X 0,Y 439.373,Z 529.753,A -85,B 0,C 180,E1 -9053.714,E2 -9053.714} C_VEL
LIN {X 0,Y 439.371,Z 529.756,A -85,B 0,C 180,E1 -9057.055,E2 -9057.055} C_VEL
LIN {X 0,Y 439.382,Z 529.755,A -85,B 0,C 180,E1 -9060.275,E2 -9060.275} C_VEL
LIN {X 0,Y 439.471,Z 529.942,A -85,B 0,C 180,E1 -9063.143,E2 -9063.143} C_VEL
LIN {X 0,Y 441.784,Z 541.193,A -85,B 0,C 180,E1 -9065.569,E2 -9065.569} C_VEL
LIN {X 0,Y 442.315,Z 544.95,A -85,B 0,C 180,E1 -9066.347,E2 -9066.347} C_VEL
LIN {X 0,Y 441.296,Z 561.188,A -85,B 0,C 180,E1 -9069.491,E2 -9069.491} C_VEL
LIN {X 0,Y 440.63,Z 573.147,A -85,B 0,C 180,E1 -9071.774,E2 -9071.774} C_VEL
LIN {X 0,Y 444.313,Z 595.505,A -85,B 0,C 180,E1 -9072.314,E2 -9072.314} C_VEL
LIN {X 0,Y 443.468,Z 680.899,A -85,B 0,C 180,E1 -9073.722,E2 -9073.722} C_VEL
LIN {X 0,Y 442.963,Z 694.266,A -85,B 0,C 180,E1 -9074.117,E2 -9074.117} C_VEL
LIN {X 0,Y 442.454,Z 707.025,A -85,B 0,C 180,E1 -9074.688,E2 -9074.688} C_VEL
LIN {X 0,Y 441.821,Z 718.368,A -85,B 0,C 180,E1 -9075.374,E2 -9075.374} C_VEL
LIN {X 0,Y 441.099,Z 730.297,A -85,B 0,C 180,E1 -9076.313,E2 -9076.313} C_VEL
LIN {X 0,Y 440.527,Z 740.558,A -85,B 0,C 180,E1 -9077.329,E2 -9077.329} C_VEL
LIN {X 0,Y 439.882,Z 750.038,A -85,B 0,C 180,E1 -9078.48,E2 -9078.48} C_VEL
LIN {X 0,Y 439.299,Z 759.172,A -85,B 0,C 180,E1 -9079.865,E2 -9079.865} C_VEL
LIN {X 0,Y 438.883,Z 766.538,A -85,B 0,C 180,E1 -9081.25,E2 -9081.25} C_VEL
LIN {X 0,Y 438.608,Z 772.455,A -85,B 0,C 180,E1 -9082.635,E2 -9082.635} C_VEL
LIN {X 0,Y 438.395,Z 776.961,A -85,B 0,C 180,E1 -9083.965,E2 -9083.965} C_VEL
LIN {X 0,Y 438.346,Z 780.699,A -85,B 0,C 180,E1 -9085.402,E2 -9085.402} C_VEL
LIN {X 0,Y 438.282,Z 782.53,A -85,B 0,C 180,E1 -9086.323,E2 -9086.323} C_VEL
LIN {X 0,Y 438.341,Z 783.908,A -85,B 0,C 180,E1 -9087.243,E2 -9087.243} C_VEL
LIN {X 0,Y 438.252,Z 785.482,A -85,B 0,C 180,E1 -9089.081,E2 -9089.081} C_VEL
LIN {X 0,Y 438.253,Z 785.675,A -85,B 0,C 180,E1 -9090,E2 -9090} C_VEL
LIN {X 0,Y 438.278,Z 784.818,A -85,B 0,C 180,E1 -9091.838,E2 -9091.838} C_VEL
LIN {X 0,Y 438.341,Z 783.809,A -85,B 0,C 180,E1 -9092.757,E2 -9092.757} C_VEL
LIN {X 0,Y 438.283,Z 782.384,A -85,B 0,C 180,E1 -9093.677,E2 -9093.677} C_VEL
LIN {X 0,Y 438.392,Z 779.418,A -85,B 0,C 180,E1 -9095.058,E2 -9095.058} C_VEL
LIN {X 0,Y 438.448,Z 775.4,A -85,B 0,C 180,E1 -9096.442,E2 -9096.442} C_VEL
LIN {X 0,Y 438.722,Z 769.216,A -85,B 0,C 180,E1 -9098.057,E2 -9098.057} C_VEL
LIN {X 0,Y 439.065,Z 762.471,A -85,B 0,C 180,E1 -9099.443,E2 -9099.443} C_VEL
LIN {X 0,Y 439.512,Z 754.097,A -85,B 0,C 180,E1 -9100.829,E2 -9100.829} C_VEL
LIN {X 0,Y 440.1,Z 745.476,A -85,B 0,C 180,E1 -9101.981,E2 -9101.981} C_VEL
LIN {X 0,Y 440.684,Z 735.182,A -85,B 0,C 180,E1 -9103.101,E2 -9103.101} C_VEL
LIN {X 0,Y 441.316,Z 724.282,A -85,B 0,C 180,E1 -9104.055,E2 -9104.055} C_VEL
LIN {X 0,Y 441.876,Z 712.589,A -85,B 0,C 180,E1 -9104.86,E2 -9104.86} C_VEL
LIN {X 0,Y 442.437,Z 700.427,A -85,B 0,C 180,E1 -9105.489,E2 -9105.489} C_VEL
LIN {X 0,Y 442.965,Z 687.178,A -85,B 0,C 180,E1 -9105.972,E2 -9105.972} C_VEL
LIN {X 0,Y 443.242,Z 674.214,A -85,B 0,C 180,E1 -9106.257,E2 -9106.257} C_VEL
LIN {X 0,Y 443.851,Z 594.955,A -85,B 0,C 180,E1 -9107.541,E2 -9107.541} C_VEL
LIN {X 0,Y 440.489,Z 573.074,A -85,B 0,C 180,E1 -9108.052,E2 -9108.052} C_VEL
LIN {X 0,Y 441.365,Z 556.236,A -85,B 0,C 180,E1 -9111.238,E2 -9111.238} C_VEL
LIN {X 0,Y 442.006,Z 543.532,A -85,B 0,C 180,E1 -9113.67,E2 -9113.67} C_VEL
LIN {X 0,Y 439.929,Z 532.041,A -85,B 0,C 180,E1 -9116.043,E2 -9116.043} C_VEL
LIN {X 0,Y 439.445,Z 529.747,A -85,B 0,C 180,E1 -9116.533,E2 -9116.533} C_VEL
LIN {X 0,Y 439.382,Z 529.756,A -85,B 0,C 180,E1 -9119.725,E2 -9119.725} C_VEL
LIN {X 0,Y 439.371,Z 529.752,A -85,B 0,C 180,E1 -9122.945,E2 -9122.945} C_VEL
LIN {X 0,Y 439.373,Z 529.75,A -85,B 0,C 180,E1 -9126.286,E2 -9126.286} C_VEL
LIN {X 0,Y 439.41,Z 529.749,A -85,B 0,C 180,E1 -9129.85,E2 -9129.85} C_VEL
LIN {X 0,Y 439.382,Z 529.749,A -85,B 0,C 180,E1 -9132.627,E2 -9132.627} C_VEL
LIN {X 0,Y 439.398,Z 529.753,A -85,B 0,C 180,E1 -9135.27,E2 -9135.27} C_VEL
LIN {X 0,Y 439.393,Z 529.748,A -85,B 0,C 180,E1 -9138.741,E2 -9138.741} C_VEL
LIN {X 0,Y 439.386,Z 529.755,A -85,B 0,C 180,E1 -9141.604,E2 -9141.604} C_VEL
LIN {X 0,Y 439.395,Z 529.749,A -85,B 0,C 180,E1 -9144.844,E2 -9144.844} C_VEL
LIN {X 0,Y 439.368,Z 529.752,A -85,B 0,C 180,E1 -9148.139,E2 -9148.139} C_VEL
LIN {X 0,Y 439.418,Z 529.751,A -85,B 0,C 180,E1 -9151.327,E2 -9151.327} C_VEL
LIN {X 0,Y 439.397,Z 529.747,A -85,B 0,C 180,E1 -9154.415,E2 -9154.415} C_VEL
LIN {X 0,Y 439.357,Z 529.76,A -85,B 0,C 180,E1 -9157.424,E2 -9157.424} C_VEL
LIN {X 0,Y 439.433,Z 529.743,A -85,B 0,C 180,E1 -9160.662,E2 -9160.662} C_VEL
LIN {X 0,Y 439.454,Z 529.74,A -85,B 0,C 180,E1 -9164.224,E2 -9164.224} C_VEL
LIN {X 0,Y 439.475,Z 529.739,A -85,B 0,C 180,E1 -9168.001,E2 -9168.001} C_VEL
LIN {X 0,Y 439.539,Z 529.734,A -85,B 0,C 180,E1 -9171.726,E2 -9171.726} C_VEL
LIN {X 0,Y 439.612,Z 529.72,A -85,B 0,C 180,E1 -9174.496,E2 -9174.496} C_VEL
LIN {X 0,Y 439.626,Z 529.719,A -85,B 0,C 180,E1 -9178.168,E2 -9178.168} C_VEL
LIN {X 0,Y 439.754,Z 529.704,A -85,B 0,C 180,E1 -9180,E2 -9180} C_VEL
LIN {X 0,Y 439.648,Z 529.717,A -85,B 0,C 180,E1 -9182.749,E2 -9182.749} C_VEL
LIN {X 0,Y 439.612,Z 529.72,A -85,B 0,C 180,E1 -9186.425,E2 -9186.425} C_VEL
LIN {X 0,Y 439.492,Z 529.74,A -85,B 0,C 180,E1 -9189.202,E2 -9189.202} C_VEL
LIN {X 0,Y 439.457,Z 529.742,A -85,B 0,C 180,E1 -9192.938,E2 -9192.938} C_VEL
LIN {X 0,Y 439.439,Z 529.742,A -85,B 0,C 180,E1 -9196.349,E2 -9196.349} C_VEL
LIN {X 0,Y 439.394,Z 529.753,A -85,B 0,C 180,E1 -9199.627,E2 -9199.627} C_VEL
LIN {X 0,Y 439.358,Z 529.752,A -85,B 0,C 180,E1 -9202.576,E2 -9202.576} C_VEL
LIN {X 0,Y 439.399,Z 529.753,A -85,B 0,C 180,E1 -9205.586,E2 -9205.586} C_VEL
LIN {X 0,Y 439.419,Z 529.745,A -85,B 0,C 180,E1 -9208.674,E2 -9208.674} C_VEL
LIN {X 0,Y 439.37,Z 529.753,A -85,B 0,C 180,E1 -9211.861,E2 -9211.861} C_VEL
LIN {X 0,Y 439.396,Z 529.752,A -85,B 0,C 180,E1 -9215.157,E2 -9215.157} C_VEL
LIN {X 0,Y 439.386,Z 529.749,A -85,B 0,C 180,E1 -9218.595,E2 -9218.595} C_VEL
LIN {X 0,Y 439.385,Z 529.755,A -85,B 0,C 180,E1 -9221.258,E2 -9221.258} C_VEL
LIN {X 0,Y 439.403,Z 529.747,A -85,B 0,C 180,E1 -9224.729,E2 -9224.729} C_VEL
LIN {X 0,Y 439.41,Z 529.749,A -85,B 0,C 180,E1 -9227.799,E2 -9227.799} C_VEL
LIN {X 0,Y 439.449,Z 529.741,A -85,B 0,C 180,E1 -9230.231,E2 -9230.231} C_VEL
LIN {X 0,Y 439.376,Z 529.754,A -85,B 0,C 180,E1 -9233.714,E2 -9233.714} C_VEL
LIN {X 0,Y 439.372,Z 529.754,A -85,B 0,C 180,E1 -9237.055,E2 -9237.055} C_VEL
LIN {X 0,Y 439.383,Z 529.749,A -85,B 0,C 180,E1 -9240.275,E2 -9240.275} C_VEL
LIN {X 0,Y 439.43,Z 529.751,A -85,B 0,C 180,E1 -9243.397,E2 -9243.397} C_VEL
LIN {X 0,Y 439.388,Z 529.748,A -85,B 0,C 180,E1 -9246.43,E2 -9246.43} C_VEL
LIN {X 0,Y 439.392,Z 529.757,A -85,B 0,C 180,E1 -9249.398,E2 -9249.398} C_VEL
LIN {X 0,Y 439.514,Z 529.891,A -85,B 0,C 180,E1 -9251.41,E2 -9251.41} C_VEL
LIN {X 0,Y 441.037,Z 538.905,A -85,B 0,C 180,E1 -9253.57,E2 -9253.57} C_VEL
LIN {X 0,Y 440.656,Z 549.496,A -85,B 0,C 180,E1 -9255.947,E2 -9255.947} C_VEL
LIN {X 0,Y 440.641,Z 549.851,A -85,B 0,C 180,E1 -9256.026,E2 -9256.026} C_VEL
LIN {X 0,Y 444.058,Z 567.857,A -85,B 0,C 180,E1 -9256.474,E2 -9256.474} C_VEL
LIN {X 0,Y 443.257,Z 655.456,A -85,B 0,C 180,E1 -9257.905,E2 -9257.905} C_VEL
LIN {X 0,Y 442.461,Z 661.253,A -85,B 0,C 180,E1 -9258.022,E2 -9258.022} C_VEL
LIN {X 0,Y 439.41,Z 670.571,A -85,B 0,C 180,E1 -9258.227,E2 -9258.227} C_VEL
LIN {X 0,Y 436.321,Z 679.669,A -85,B 0,C 180,E1 -9258.534,E2 -9258.534} C_VEL
LIN {X 0,Y 435.465,Z 685.112,A -85,B 0,C 180,E1 -9258.807,E2 -9258.807} C_VEL
LIN {X 0,Y 434.904,Z 696.155,A -85,B 0,C 180,E1 -9259.526,E2 -9259.526} C_VEL
LIN {X 0,Y 434.307,Z 707.33,A -85,B 0,C 180,E1 -9260.453,E2 -9260.453} C_VEL
LIN {X 0,Y 433.585,Z 716.604,A -85,B 0,C 180,E1 -9261.401,E2 -9261.401} C_VEL
LIN {X 0,Y 433.012,Z 725.692,A -85,B 0,C 180,E1 -9262.54,E2 -9262.54} C_VEL
LIN {X 0,Y 432.715,Z 733.313,A -85,B 0,C 180,E1 -9263.706,E2 -9263.706} C_VEL
LIN {X 0,Y 432.183,Z 740.795,A -85,B 0,C 180,E1 -9265.103,E2 -9265.103} C_VEL
LIN {X 0,Y 431.781,Z 747.71,A -85,B 0,C 180,E1 -9266.734,E2 -9266.734} C_VEL
LIN {X 0,Y 431.378,Z 752.301,A -85,B 0,C 180,E1 -9268.133,E2 -9268.133} C_VEL
LIN {X 0,Y 431.278,Z 754.738,A -85,B 0,C 180,E1 -9269.066,E2 -9269.066} C_VEL
LIN {X 0,Y 431.212,Z 756.722,A -85,B 0,C 180,E1 -9270,E2 -9270} C_VEL
LIN {X 0,Y 431.196,Z 758.295,A -85,B 0,C 180,E1 -9270.934,E2 -9270.934} C_VEL
LIN {X 0,Y 431.223,Z 759.464,A -85,B 0,C 180,E1 -9271.868,E2 -9271.868} C_VEL
LIN {X 0,Y 431.27,Z 760.197,A -85,B 0,C 180,E1 -9272.802,E2 -9272.802} C_VEL
LIN {X 0,Y 431.201,Z 760.521,A -85,B 0,C 180,E1 -9274.674,E2 -9274.674} C_VEL
LIN {X 0,Y 431.247,Z 759.603,A -85,B 0,C 180,E1 -9276.217,E2 -9276.217} C_VEL
LIN {X 0,Y 431.281,Z 758.013,A -85,B 0,C 180,E1 -9277.491,E2 -9277.491} C_VEL
LIN {X 0,Y 431.369,Z 755.362,A -85,B 0,C 180,E1 -9278.904,E2 -9278.904} C_VEL
LIN {X 0,Y 431.511,Z 751.691,A -85,B 0,C 180,E1 -9280.32,E2 -9280.32} C_VEL
LIN {X 0,Y 431.851,Z 746.889,A -85,B 0,C 180,E1 -9281.737,E2 -9281.737} C_VEL
LIN {X 0,Y 432.209,Z 740.81,A -85,B 0,C 180,E1 -9283.158,E2 -9283.158} C_VEL
LIN {X 0,Y 432.731,Z 733.231,A -85,B 0,C 180,E1 -9284.58,E2 -9284.58} C_VEL
LIN {X 0,Y 433.308,Z 725.454,A -85,B 0,C 180,E1 -9285.764,E2 -9285.764} C_VEL
LIN {X 0,Y 434.003,Z 715.267,A -85,B 0,C 180,E1 -9287.02,E2 -9287.02} C_VEL
LIN {X 0,Y 434.722,Z 704.015,A -85,B 0,C 180,E1 -9288.132,E2 -9288.132} C_VEL
LIN {X 0,Y 435.383,Z 693.427,A -85,B 0,C 180,E1 -9288.957,E2 -9288.957} C_VEL
LIN {X 0,Y 436,Z 680.63,A -85,B 0,C 180,E1 -9289.724,E2 -9289.724} C_VEL
LIN {X 0,Y 436.515,Z 667.747,A -85,B 0,C 180,E1 -9290.283,E2 -9290.283} C_VEL
LIN {X 0,Y 436.818,Z 655.088,A -85,B 0,C 180,E1 -9290.637,E2 -9290.637} C_VEL
LIN {X 0,Y 437.699,Z 568.488,A -85,B 0,C 180,E1 -9292.083,E2 -9292.083} C_VEL
LIN {X 0,Y 433.933,Z 550.139,A -85,B 0,C 180,E1 -9292.59,E2 -9292.59} C_VEL
LIN {X 0,Y 434.324,Z 541.32,A -85,B 0,C 180,E1 -9294.624,E2 -9294.624} C_VEL
LIN {X 0,Y 432.518,Z 531.05,A -85,B 0,C 180,E1 -9297.193,E2 -9297.193} C_VEL
LIN {X 0,Y 432.436,Z 530.621,A -85,B 0,C 180,E1 -9297.33,E2 -9297.33} C_VEL
LIN {X 0,Y 432.348,Z 530.625,A -85,B 0,C 180,E1 -9300.51,E2 -9300.51} C_VEL
LIN {X 0,Y 432.359,Z 530.628,A -85,B 0,C 180,E1 -9304.003,E2 -9304.003} C_VEL
LIN {X 0,Y 432.333,Z 530.63,A -85,B 0,C 180,E1 -9307.198,E2 -9307.198} C_VEL
LIN {X 0,Y 432.356,Z 530.629,A -85,B 0,C 180,E1 -9310.182,E2 -9310.182} C_VEL
LIN {X 0,Y 432.363,Z 530.627,A -85,B 0,C 180,E1 -9313.054,E2 -9313.054} C_VEL
LIN {X 0,Y 432.338,Z 530.627,A -85,B 0,C 180,E1 -9315.663,E2 -9315.663} C_VEL
LIN {X 0,Y 432.363,Z 530.624,A -85,B 0,C 180,E1 -9318.392,E2 -9318.392} C_VEL
LIN {X 0,Y 432.344,Z 530.628,A -85,B 0,C 180,E1 -9321.85,E2 -9321.85} C_VEL
LIN {X 0,Y 432.336,Z 530.628,A -85,B 0,C 180,E1 -9325.322,E2 -9325.322} C_VEL
LIN {X 0,Y 432.321,Z 530.634,A -85,B 0,C 180,E1 -9328.654,E2 -9328.654} C_VEL
LIN {X 0,Y 432.375,Z 530.624,A -85,B 0,C 180,E1 -9331.368,E2 -9331.368} C_VEL
LIN {X 0,Y 432.358,Z 530.622,A -85,B 0,C 180,E1 -9333.967,E2 -9333.967} C_VEL
LIN {X 0,Y 432.312,Z 530.629,A -85,B 0,C 180,E1 -9337.035,E2 -9337.035} C_VEL
LIN {X 0,Y 432.379,Z 530.629,A -85,B 0,C 180,E1 -9340.514,E2 -9340.514} C_VEL
LIN {X 0,Y 432.422,Z 530.617,A -85,B 0,C 180,E1 -9343.961,E2 -9343.961} C_VEL
LIN {X 0,Y 432.451,Z 530.609,A -85,B 0,C 180,E1 -9347.803,E2 -9347.803} C_VEL
LIN {X 0,Y 432.483,Z 530.606,A -85,B 0,C 180,E1 -9351.59,E2 -9351.59} C_VEL
LIN {X 0,Y 432.591,Z 530.599,A -85,B 0,C 180,E1 -9354.406,E2 -9354.406} C_VEL
LIN {X 0,Y 432.597,Z 530.592,A -85,B 0,C 180,E1 -9358.138,E2 -9358.138} C_VEL
LIN {X 0,Y 432.725,Z 530.58,A -85,B 0,C 180,E1 -9360,E2 -9360} C_VEL
LIN {X 0,Y 432.597,Z 530.594,A -85,B 0,C 180,E1 -9362.793,E2 -9362.793} C_VEL
LIN {X 0,Y 432.563,Z 530.606,A -85,B 0,C 180,E1 -9366.53,E2 -9366.53} C_VEL
LIN {X 0,Y 432.435,Z 530.614,A -85,B 0,C 180,E1 -9369.353,E2 -9369.353} C_VEL
LIN {X 0,Y 432.422,Z 530.616,A -85,B 0,C 180,E1 -9372.804,E2 -9372.804} C_VEL
LIN {X 0,Y 432.404,Z 530.626,A -85,B 0,C 180,E1 -9376.479,E2 -9376.479} C_VEL
LIN {X 0,Y 432.33,Z 530.628,A -85,B 0,C 180,E1 -9379.961,E2 -9379.961} C_VEL
LIN {X 0,Y 432.311,Z 530.631,A -85,B 0,C 180,E1 -9382.965,E2 -9382.965} C_VEL
LIN {X 0,Y 432.357,Z 530.627,A -85,B 0,C 180,E1 -9386.033,E2 -9386.033} C_VEL
LIN {X 0,Y 432.345,Z 530.628,A -85,B 0,C 180,E1 -9389.187,E2 -9389.187} C_VEL
LIN {X 0,Y 432.319,Z 530.634,A -85,B 0,C 180,E1 -9392.294,E2 -9392.294} C_VEL
LIN {X 0,Y 432.335,Z 530.634,A -85,B 0,C 180,E1 -9394.678,E2 -9394.678} C_VEL
LIN {X 0,Y 432.346,Z 530.629,A -85,B 0,C 180,E1 -9398.149,E2 -9398.149} C_VEL
LIN {X 0,Y 432.361,Z 530.626,A -85,B 0,C 180,E1 -9401.608,E2 -9401.608} C_VEL
LIN {X 0,Y 432.329,Z 530.635,A -85,B 0,C 180,E1 -9404.348,E2 -9404.348} C_VEL
LIN {X 0,Y 432.321,Z 530.633,A -85,B 0,C 180,E1 -9407.016,E2 -9407.016} C_VEL
LIN {X 0,Y 432.338,Z 530.629,A -85,B 0,C 180,E1 -9409.82,E2 -9409.82} C_VEL
LIN {X 0,Y 432.312,Z 530.634,A -85,B 0,C 180,E1 -9413.024,E2 -9413.024} C_VEL
LIN {X 0,Y 432.357,Z 530.628,A -85,B 0,C 180,E1 -9415.997,E2 -9415.997} C_VEL
LIN {X 0,Y 432.347,Z 530.629,A -85,B 0,C 180,E1 -9419.49,E2 -9419.49} C_VEL
LIN {X 0,Y 432.429,Z 530.682,A -85,B 0,C 180,E1 -9422.833,E2 -9422.833} C_VEL
LIN {X 0,Y 435.045,Z 543.638,A -85,B 0,C 180,E1 -9425.674,E2 -9425.674} C_VEL
LIN {X 0,Y 435.347,Z 547.366,A -85,B 0,C 180,E1 -9426.446,E2 -9426.446} C_VEL
LIN {X 0,Y 434.24,Z 563.343,A -85,B 0,C 180,E1 -9429.587,E2 -9429.587} C_VEL
LIN {X 0,Y 433.694,Z 572.879,A -85,B 0,C 180,E1 -9431.444,E2 -9431.444} C_VEL
LIN {X 0,Y 437.583,Z 596.535,A -85,B 0,C 180,E1 -9432.033,E2 -9432.033} C_VEL
LIN {X 0,Y 436.685,Z 681.48,A -85,B 0,C 180,E1 -9433.462,E2 -9433.462} C_VEL
LIN {X 0,Y 436.11,Z 695.337,A -85,B 0,C 180,E1 -9433.89,E2 -9433.89} C_VEL
LIN {X 0,Y 435.57,Z 708.258,A -85,B 0,C 180,E1 -9434.5,E2 -9434.5} C_VEL
LIN {X 0,Y 434.836,Z 720.015,A -85,B 0,C 180,E1 -9435.253,E2 -9435.253} C_VEL
LIN {X 0,Y 434.184,Z 730.604,A -85,B 0,C 180,E1 -9436.118,E2 -9436.118} C_VEL
LIN {X 0,Y 433.526,Z 741.587,A -85,B 0,C 180,E1 -9437.24,E2 -9437.24} C_VEL
LIN {X 0,Y 432.77,Z 751.604,A -85,B 0,C 180,E1 -9438.526,E2 -9438.526} C_VEL
LIN {X 0,Y 432.201,Z 760.431,A -85,B 0,C 180,E1 -9439.933,E2 -9439.933} C_VEL
LIN {X 0,Y 431.79,Z 767.513,A -85,B 0,C 180,E1 -9441.341,E2 -9441.341} C_VEL
LIN {X 0,Y 431.434,Z 773.983,A -85,B 0,C 180,E1 -9442.983,E2 -9442.983} C_VEL
LIN {X 0,Y 431.295,Z 778.263,A -85,B 0,C 180,E1 -9444.389,E2 -9444.389} C_VEL
LIN {X 0,Y 431.276,Z 780.534,A -85,B 0,C 180,E1 -9445.327,E2 -9445.327} C_VEL
LIN {X 0,Y 431.189,Z 782.352,A -85,B 0,C 180,E1 -9446.262,E2 -9446.262} C_VEL
LIN {X 0,Y 431.236,Z 783.724,A -85,B 0,C 180,E1 -9447.198,E2 -9447.198} C_VEL
LIN {X 0,Y 431.202,Z 784.699,A -85,B 0,C 180,E1 -9448.132,E2 -9448.132} C_VEL
LIN {X 0,Y 431.168,Z 785.287,A -85,B 0,C 180,E1 -9449.066,E2 -9449.066} C_VEL
LIN {X 0,Y 431.167,Z 785.468,A -85,B 0,C 180,E1 -9450,E2 -9450} C_VEL
LIN {X 0,Y 431.202,Z 784.599,A -85,B 0,C 180,E1 -9451.868,E2 -9451.868} C_VEL
LIN {X 0,Y 431.236,Z 783.583,A -85,B 0,C 180,E1 -9452.802,E2 -9452.802} C_VEL
LIN {X 0,Y 431.19,Z 782.147,A -85,B 0,C 180,E1 -9453.738,E2 -9453.738} C_VEL
LIN {X 0,Y 431.303,Z 779.17,A -85,B 0,C 180,E1 -9455.142,E2 -9455.142} C_VEL
LIN {X 0,Y 431.377,Z 775.138,A -85,B 0,C 180,E1 -9456.548,E2 -9456.548} C_VEL
LIN {X 0,Y 431.656,Z 768.933,A -85,B 0,C 180,E1 -9458.19,E2 -9458.19} C_VEL
LIN {X 0,Y 432.012,Z 762.169,A -85,B 0,C 180,E1 -9459.599,E2 -9459.599} C_VEL
LIN {X 0,Y 432.485,Z 753.768,A -85,B 0,C 180,E1 -9461.007,E2 -9461.007} C_VEL
LIN {X 0,Y 433.112,Z 745.113,A -85,B 0,C 180,E1 -9462.178,E2 -9462.178} C_VEL
LIN {X 0,Y 433.721,Z 735.239,A -85,B 0,C 180,E1 -9463.269,E2 -9463.269} C_VEL
LIN {X 0,Y 434.392,Z 723.842,A -85,B 0,C 180,E1 -9464.284,E2 -9464.284} C_VEL
LIN {X 0,Y 435.007,Z 712.055,A -85,B 0,C 180,E1 -9465.1,E2 -9465.1} C_VEL
LIN {X 0,Y 435.554,Z 699.786,A -85,B 0,C 180,E1 -9465.74,E2 -9465.74} C_VEL
LIN {X 0,Y 436.091,Z 687.278,A -85,B 0,C 180,E1 -9466.2,E2 -9466.2} C_VEL
LIN {X 0,Y 436.373,Z 674.599,A -85,B 0,C 180,E1 -9466.49,E2 -9466.49} C_VEL
LIN {X 0,Y 437.001,Z 595.479,A -85,B 0,C 180,E1 -9467.792,E2 -9467.792} C_VEL
LIN {X 0,Y 433.529,Z 572.868,A -85,B 0,C 180,E1 -9468.329,E2 -9468.329} C_VEL
LIN {X 0,Y 434.447,Z 555.927,A -85,B 0,C 180,E1 -9471.593,E2 -9471.593} C_VEL
LIN {X 0,Y 435.059,Z 545.773,A -85,B 0,C 180,E1 -9473.566,E2 -9473.566} C_VEL
LIN {X 0,Y 434.084,Z 539.068,A -85,B 0,C 180,E1 -9474.951,E2 -9474.951} C_VEL
LIN {X 0,Y 432.414,Z 530.622,A -85,B 0,C 180,E1 -9476.801,E2 -9476.801} C_VEL
LIN {X 0,Y 432.344,Z 530.63,A -85,B 0,C 180,E1 -9480.259,E2 -9480.259} C_VEL
LIN {X 0,Y 432.338,Z 530.634,A -85,B 0,C 180,E1 -9483.551,E2 -9483.551} C_VEL
LIN {X 0,Y 432.337,Z 530.63,A -85,B 0,C 180,E1 -9485.817,E2 -9485.817} C_VEL
LIN {X 0,Y 432.353,Z 530.631,A -85,B 0,C 180,E1 -9489.341,E2 -9489.341} C_VEL
LIN {X 0,Y 432.332,Z 530.631,A -85,B 0,C 180,E1 -9491.796,E2 -9491.796} C_VEL
LIN {X 0,Y 432.336,Z 530.627,A -85,B 0,C 180,E1 -9494.346,E2 -9494.346} C_VEL
LIN {X 0,Y 432.315,Z 530.632,A -85,B 0,C 180,E1 -9497.015,E2 -9497.015} C_VEL
LIN {X 0,Y 432.351,Z 530.628,A -85,B 0,C 180,E1 -9499.816,E2 -9499.816} C_VEL
LIN {X 0,Y 432.311,Z 530.633,A -85,B 0,C 180,E1 -9503.022,E2 -9503.022} C_VEL
LIN {X 0,Y 432.353,Z 530.626,A -85,B 0,C 180,E1 -9505.996,E2 -9505.996} C_VEL
LIN {X 0,Y 432.388,Z 530.625,A -85,B 0,C 180,E1 -9509.743,E2 -9509.743} C_VEL
LIN {X 0,Y 432.393,Z 530.627,A -85,B 0,C 180,E1 -9513.372,E2 -9513.372} C_VEL
LIN {X 0,Y 432.363,Z 530.625,A -85,B 0,C 180,E1 -9516.023,E2 -9516.023} C_VEL
LIN {X 0,Y 432.342,Z 530.629,A -85,B 0,C 180,E1 -9519.046,E2 -9519.046} C_VEL
LIN {X 0,Y 432.369,Z 530.624,A -85,B 0,C 180,E1 -9522.011,E2 -9522.011} C_VEL
LIN {X 0,Y 432.387,Z 530.622,A -85,B 0,C 180,E1 -9524.926,E2 -9524.926} C_VEL
LIN {X 0,Y 432.45,Z 530.616,A -85,B 0,C 180,E1 -9527.803,E2 -9527.803} C_VEL
LIN {X 0,Y 432.483,Z 530.614,A -85,B 0,C 180,E1 -9531.59,E2 -9531.59} C_VEL
LIN {X 0,Y 432.589,Z 530.595,A -85,B 0,C 180,E1 -9534.406,E2 -9534.406} C_VEL
LIN {X 0,Y 432.596,Z 530.595,A -85,B 0,C 180,E1 -9538.138,E2 -9538.138} C_VEL
LIN {X 0,Y 432.724,Z 530.58,A -85,B 0,C 180,E1 -9540,E2 -9540} C_VEL
LIN {X 0,Y 432.598,Z 530.595,A -85,B 0,C 180,E1 -9542.794,E2 -9542.794} C_VEL
LIN {X 0,Y 432.566,Z 530.598,A -85,B 0,C 180,E1 -9546.531,E2 -9546.531} C_VEL
LIN {X 0,Y 432.435,Z 530.622,A -85,B 0,C 180,E1 -9549.353,E2 -9549.353} C_VEL
LIN {X 0,Y 432.422,Z 530.617,A -85,B 0,C 180,E1 -9552.804,E2 -9552.804} C_VEL
LIN {X 0,Y 432.404,Z 530.618,A -85,B 0,C 180,E1 -9556.479,E2 -9556.479} C_VEL
LIN {X 0,Y 432.331,Z 530.629,A -85,B 0,C 180,E1 -9559.961,E2 -9559.961} C_VEL
LIN {X 0,Y 432.312,Z 530.632,A -85,B 0,C 180,E1 -9562.965,E2 -9562.965} C_VEL
LIN {X 0,Y 432.358,Z 530.625,A -85,B 0,C 180,E1 -9566.033,E2 -9566.033} C_VEL
LIN {X 0,Y 432.346,Z 530.63,A -85,B 0,C 180,E1 -9569.188,E2 -9569.188} C_VEL
LIN {X 0,Y 432.32,Z 530.629,A -85,B 0,C 180,E1 -9572.294,E2 -9572.294} C_VEL
LIN {X 0,Y 432.336,Z 530.627,A -85,B 0,C 180,E1 -9574.678,E2 -9574.678} C_VEL
LIN {X 0,Y 432.343,Z 530.627,A -85,B 0,C 180,E1 -9578.15,E2 -9578.15} C_VEL
LIN {X 0,Y 432.33,Z 530.633,A -85,B 0,C 180,E1 -9581.603,E2 -9581.603} C_VEL
LIN {X 0,Y 432.338,Z 530.627,A -85,B 0,C 180,E1 -9584.347,E2 -9584.347} C_VEL
LIN {X 0,Y 432.363,Z 530.626,A -85,B 0,C 180,E1 -9587.01,E2 -9587.01} C_VEL
LIN {X 0,Y 432.356,Z 530.627,A -85,B 0,C 180,E1 -9589.818,E2 -9589.818} C_VEL
LIN {X 0,Y 432.315,Z 530.633,A -85,B 0,C 180,E1 -9593.024,E2 -9593.024} C_VEL
LIN {X 0,Y 432.359,Z 530.625,A -85,B 0,C 180,E1 -9595.997,E2 -9595.997} C_VEL
LIN {X 0,Y 432.348,Z 530.632,A -85,B 0,C 180,E1 -9599.49,E2 -9599.49} C_VEL
LIN {X 0,Y 432.392,Z 530.622,A -85,B 0,C 180,E1 -9602.929,E2 -9602.929} C_VEL
LIN {X 0,Y 432.373,Z 530.623,A -85,B 0,C 180,E1 -9606.024,E2 -9606.024} C_VEL
LIN {X 0,Y 432.353,Z 530.634,A -85,B 0,C 180,E1 -9609.047,E2 -9609.047} C_VEL
LIN {X 0,Y 432.472,Z 530.793,A -85,B 0,C 180,E1 -9611.218,E2 -9611.218} C_VEL
LIN {X 0,Y 434.086,Z 540.335,A -85,B 0,C 180,E1 -9613.541,E2 -9613.541} C_VEL
LIN {X 0,Y 433.727,Z 550.311,A -85,B 0,C 180,E1 -9615.771,E2 -9615.771} C_VEL
LIN {X 0,Y 437.261,Z 568.668,A -85,B 0,C 180,E1 -9616.223,E2 -9616.223} C_VEL
LIN {X 0,Y 436.368,Z 657.542,A -85,B 0,C 180,E1 -9617.708,E2 -9617.708} C_VEL
LIN {X 0,Y 435.99,Z 671.257,A -85,B 0,C 180,E1 -9618.14,E2 -9618.14} C_VEL
LIN {X 0,Y 435.528,Z 683.571,A -85,B 0,C 180,E1 -9618.717,E2 -9618.717} C_VEL
LIN {X 0,Y 435.465,Z 685.112,A -85,B 0,C 180,E1 -9618.807,E2 -9618.807} C_VEL
LIN {X 0,Y 434.593,Z 690.564,A -85,B 0,C 180,E1 -9619.117,E2 -9619.117} C_VEL
LIN {X 0,Y 431.361,Z 699.132,A -85,B 0,C 180,E1 -9619.635,E2 -9619.635} C_VEL
LIN {X 0,Y 428.037,Z 707.236,A -85,B 0,C 180,E1 -9620.242,E2 -9620.242} C_VEL
LIN {X 0,Y 427.016,Z 711.941,A -85,B 0,C 180,E1 -9620.684,E2 -9620.684} C_VEL
LIN {X 0,Y 426.454,Z 721.093,A -85,B 0,C 180,E1 -9621.732,E2 -9621.732} C_VEL
LIN {X 0,Y 425.961,Z 729.424,A -85,B 0,C 180,E1 -9622.892,E2 -9622.892} C_VEL
LIN {X 0,Y 425.325,Z 737.706,A -85,B 0,C 180,E1 -9624.31,E2 -9624.31} C_VEL
LIN {X 0,Y 424.897,Z 744.378,A -85,B 0,C 180,E1 -9625.732,E2 -9625.732} C_VEL
LIN {X 0,Y 424.48,Z 749.717,A -85,B 0,C 180,E1 -9627.153,E2 -9627.153} C_VEL
LIN {X 0,Y 424.344,Z 753.885,A -85,B 0,C 180,E1 -9628.576,E2 -9628.576} C_VEL
LIN {X 0,Y 424.126,Z 757.015,A -85,B 0,C 180,E1 -9630,E2 -9630} C_VEL
LIN {X 0,Y 424.114,Z 758.572,A -85,B 0,C 180,E1 -9630.949,E2 -9630.949} C_VEL
LIN {X 0,Y 424.149,Z 759.713,A -85,B 0,C 180,E1 -9631.899,E2 -9631.899} C_VEL
LIN {X 0,Y 424.164,Z 760.426,A -85,B 0,C 180,E1 -9632.849,E2 -9632.849} C_VEL
LIN {X 0,Y 424.127,Z 760.718,A -85,B 0,C 180,E1 -9634.752,E2 -9634.752} C_VEL
LIN {X 0,Y 424.167,Z 759.865,A -85,B 0,C 180,E1 -9636.204,E2 -9636.204} C_VEL
LIN {X 0,Y 424.198,Z 758.145,A -85,B 0,C 180,E1 -9637.616,E2 -9637.616} C_VEL
LIN {X 0,Y 424.318,Z 755.46,A -85,B 0,C 180,E1 -9639.053,E2 -9639.053} C_VEL
LIN {X 0,Y 424.483,Z 751.753,A -85,B 0,C 180,E1 -9640.493,E2 -9640.493} C_VEL
LIN {X 0,Y 424.815,Z 746.913,A -85,B 0,C 180,E1 -9641.934,E2 -9641.934} C_VEL
LIN {X 0,Y 425.212,Z 740.792,A -85,B 0,C 180,E1 -9643.379,E2 -9643.379} C_VEL
LIN {X 0,Y 425.791,Z 733.158,A -85,B 0,C 180,E1 -9644.823,E2 -9644.823} C_VEL
LIN {X 0,Y 426.424,Z 725.313,A -85,B 0,C 180,E1 -9646.025,E2 -9646.025} C_VEL
LIN {X 0,Y 427.096,Z 715.704,A -85,B 0,C 180,E1 -9647.229,E2 -9647.229} C_VEL
LIN {X 0,Y 427.813,Z 705.009,A -85,B 0,C 180,E1 -9648.311,E2 -9648.311} C_VEL
LIN {X 0,Y 428.512,Z 694.649,A -85,B 0,C 180,E1 -9649.148,E2 -9649.148} C_VEL
LIN {X 0,Y 429.149,Z 683.365,A -85,B 0,C 180,E1 -9649.865,E2 -9649.865} C_VEL
LIN {X 0,Y 429.647,Z 670.602,A -85,B 0,C 180,E1 -9650.465,E2 -9650.465} C_VEL
LIN {X 0,Y 430.074,Z 657.286,A -85,B 0,C 180,E1 -9650.882,E2 -9650.882} C_VEL
LIN {X 0,Y 431.001,Z 569.395,A -85,B 0,C 180,E1 -9652.383,E2 -9652.383} C_VEL
LIN {X 0,Y 427.087,Z 550.284,A -85,B 0,C 180,E1 -9652.934,E2 -9652.934} C_VEL
LIN {X 0,Y 427.388,Z 542.674,A -85,B 0,C 180,E1 -9654.721,E2 -9654.721} C_VEL
LIN {X 0,Y 425.7,Z 533.104,A -85,B 0,C 180,E1 -9657.15,E2 -9657.15} C_VEL
LIN {X 0,Y 425.374,Z 531.498,A -85,B 0,C 180,E1 -9657.622,E2 -9657.622} C_VEL
LIN {X 0,Y 425.288,Z 531.504,A -85,B 0,C 180,E1 -9660.815,E2 -9660.815} C_VEL
LIN {X 0,Y 425.311,Z 531.509,A -85,B 0,C 180,E1 -9664.287,E2 -9664.287} C_VEL
LIN {X 0,Y 425.287,Z 531.505,A -85,B 0,C 180,E1 -9667.692,E2 -9667.692} C_VEL
LIN {X 0,Y 425.301,Z 531.51,A -85,B 0,C 180,E1 -9670.523,E2 -9670.523} C_VEL
LIN {X 0,Y 425.314,Z 531.503,A -85,B 0,C 180,E1 -9673.358,E2 -9673.358} C_VEL
LIN {X 0,Y 425.261,Z 531.516,A -85,B 0,C 180,E1 -9676.647,E2 -9676.647} C_VEL
LIN {X 0,Y 425.301,Z 531.499,A -85,B 0,C 180,E1 -9679.874,E2 -9679.874} C_VEL
LIN {X 0,Y 425.28,Z 531.512,A -85,B 0,C 180,E1 -9682.486,E2 -9682.486} C_VEL
LIN {X 0,Y 425.302,Z 531.503,A -85,B 0,C 180,E1 -9685.817,E2 -9685.817} C_VEL
LIN {X 0,Y 425.296,Z 531.502,A -85,B 0,C 180,E1 -9689.235,E2 -9689.235} C_VEL
LIN {X 0,Y 425.344,Z 531.504,A -85,B 0,C 180,E1 -9692.442,E2 -9692.442} C_VEL
LIN {X 0,Y 425.344,Z 531.499,A -85,B 0,C 180,E1 -9695.601,E2 -9695.601} C_VEL
LIN {X 0,Y 425.285,Z 531.509,A -85,B 0,C 180,E1 -9698.681,E2 -9698.681} C_VEL
LIN {X 0,Y 425.325,Z 531.498,A -85,B 0,C 180,E1 -9701.702,E2 -9701.702} C_VEL
LIN {X 0,Y 425.34,Z 531.506,A -85,B 0,C 180,E1 -9704.67,E2 -9704.67} C_VEL
LIN {X 0,Y 425.403,Z 531.486,A -85,B 0,C 180,E1 -9707.598,E2 -9707.598} C_VEL
LIN {X 0,Y 425.434,Z 531.485,A -85,B 0,C 180,E1 -9711.45,E2 -9711.45} C_VEL
LIN {X 0,Y 425.547,Z 531.475,A -85,B 0,C 180,E1 -9714.313,E2 -9714.313} C_VEL
LIN {X 0,Y 425.567,Z 531.467,A -85,B 0,C 180,E1 -9718.107,E2 -9718.107} C_VEL
LIN {X 0,Y 425.695,Z 531.455,A -85,B 0,C 180,E1 -9720,E2 -9720} C_VEL
LIN {X 0,Y 425.549,Z 531.471,A -85,B 0,C 180,E1 -9722.84,E2 -9722.84} C_VEL
LIN {X 0,Y 425.52,Z 531.482,A -85,B 0,C 180,E1 -9726.639,E2 -9726.639} C_VEL
LIN {X 0,Y 425.393,Z 531.49,A -85,B 0,C 180,E1 -9729.509,E2 -9729.509} C_VEL
LIN {X 0,Y 425.384,Z 531.491,A -85,B 0,C 180,E1 -9732.904,E2 -9732.904} C_VEL
LIN {X 0,Y 425.353,Z 531.503,A -85,B 0,C 180,E1 -9736.605,E2 -9736.605} C_VEL
LIN {X 0,Y 425.32,Z 531.5,A -85,B 0,C 180,E1 -9739.636,E2 -9739.636} C_VEL
LIN {X 0,Y 425.28,Z 531.51,A -85,B 0,C 180,E1 -9742.339,E2 -9742.339} C_VEL
LIN {X 0,Y 425.287,Z 531.506,A -85,B 0,C 180,E1 -9745.446,E2 -9745.446} C_VEL
LIN {X 0,Y 425.331,Z 531.505,A -85,B 0,C 180,E1 -9748.632,E2 -9748.632} C_VEL
LIN {X 0,Y 425.259,Z 531.51,A -85,B 0,C 180,E1 -9751.927,E2 -9751.927} C_VEL
LIN {X 0,Y 425.294,Z 531.505,A -85,B 0,C 180,E1 -9755.336,E2 -9755.336} C_VEL
LIN {X 0,Y 425.307,Z 531.506,A -85,B 0,C 180,E1 -9759.047,E2 -9759.047} C_VEL
LIN {X 0,Y 425.31,Z 531.505,A -85,B 0,C 180,E1 -9761.963,E2 -9761.963} C_VEL
LIN {X 0,Y 425.285,Z 531.508,A -85,B 0,C 180,E1 -9765.283,E2 -9765.283} C_VEL
LIN {X 0,Y 425.273,Z 531.514,A -85,B 0,C 180,E1 -9768.622,E2 -9768.622} C_VEL
LIN {X 0,Y 425.313,Z 531.506,A -85,B 0,C 180,E1 -9771.104,E2 -9771.104} C_VEL
LIN {X 0,Y 425.298,Z 531.509,A -85,B 0,C 180,E1 -9774.665,E2 -9774.665} C_VEL
LIN {X 0,Y 425.264,Z 531.514,A -85,B 0,C 180,E1 -9778.074,E2 -9778.074} C_VEL
LIN {X 0,Y 425.331,Z 531.504,A -85,B 0,C 180,E1 -9781.369,E2 -9781.369} C_VEL
LIN {X 0,Y 425.387,Z 531.531,A -85,B 0,C 180,E1 -9782.536,E2 -9782.536} C_VEL
LIN {X 0,Y 428.086,Z 544.832,A -85,B 0,C 180,E1 -9785.511,E2 -9785.511} C_VEL
LIN {X 0,Y 428.426,Z 548.829,A -85,B 0,C 180,E1 -9786.355,E2 -9786.355} C_VEL
LIN {X 0,Y 427.334,Z 563.775,A -85,B 0,C 180,E1 -9789.344,E2 -9789.344} C_VEL
LIN {X 0,Y 426.822,Z 572.591,A -85,B 0,C 180,E1 -9791.095,E2 -9791.095} C_VEL
LIN {X 0,Y 430.665,Z 595.728,A -85,B 0,C 180,E1 -9791.701,E2 -9791.701} C_VEL
LIN {X 0,Y 430.758,Z 602.966,A -85,B 0,C 180,E1 -9791.831,E2 -9791.831} C_VEL
LIN {X 0,Y 429.953,Z 680.948,A -85,B 0,C 180,E1 -9793.165,E2 -9793.165} C_VEL
LIN {X 0,Y 429.396,Z 694.151,A -85,B 0,C 180,E1 -9793.57,E2 -9793.57} C_VEL
LIN {X 0,Y 428.874,Z 706.265,A -85,B 0,C 180,E1 -9794.13,E2 -9794.13} C_VEL
LIN {X 0,Y 428.086,Z 718.508,A -85,B 0,C 180,E1 -9794.893,E2 -9794.893} C_VEL
LIN {X 0,Y 427.328,Z 729.933,A -85,B 0,C 180,E1 -9795.826,E2 -9795.826} C_VEL
LIN {X 0,Y 426.639,Z 740.507,A -85,B 0,C 180,E1 -9796.909,E2 -9796.909} C_VEL
LIN {X 0,Y 425.962,Z 749.907,A -85,B 0,C 180,E1 -9798.098,E2 -9798.098} C_VEL
LIN {X 0,Y 425.244,Z 758.982,A -85,B 0,C 180,E1 -9799.526,E2 -9799.526} C_VEL
LIN {X 0,Y 424.806,Z 766.307,A -85,B 0,C 180,E1 -9800.958,E2 -9800.958} C_VEL
LIN {X 0,Y 424.478,Z 772.189,A -85,B 0,C 180,E1 -9802.389,E2 -9802.389} C_VEL
LIN {X 0,Y 424.249,Z 776.453,A -85,B 0,C 180,E1 -9803.693,E2 -9803.693} C_VEL
LIN {X 0,Y 424.205,Z 780.372,A -85,B 0,C 180,E1 -9805.248,E2 -9805.248} C_VEL
LIN {X 0,Y 424.101,Z 782.177,A -85,B 0,C 180,E1 -9806.199,E2 -9806.199} C_VEL
LIN {X 0,Y 424.131,Z 783.541,A -85,B 0,C 180,E1 -9807.151,E2 -9807.151} C_VEL
LIN {X 0,Y 424.129,Z 784.511,A -85,B 0,C 180,E1 -9808.101,E2 -9808.101} C_VEL
LIN {X 0,Y 424.088,Z 785.092,A -85,B 0,C 180,E1 -9809.05,E2 -9809.05} C_VEL
LIN {X 0,Y 424.084,Z 785.261,A -85,B 0,C 180,E1 -9810,E2 -9810} C_VEL
LIN {X 0,Y 424.129,Z 784.38,A -85,B 0,C 180,E1 -9811.899,E2 -9811.899} C_VEL
LIN {X 0,Y 424.133,Z 783.356,A -85,B 0,C 180,E1 -9812.849,E2 -9812.849} C_VEL
LIN {X 0,Y 424.101,Z 781.906,A -85,B 0,C 180,E1 -9813.801,E2 -9813.801} C_VEL
LIN {X 0,Y 424.216,Z 778.918,A -85,B 0,C 180,E1 -9815.228,E2 -9815.228} C_VEL
LIN {X 0,Y 424.301,Z 774.87,A -85,B 0,C 180,E1 -9816.658,E2 -9816.658} C_VEL
LIN {X 0,Y 424.604,Z 768.644,A -85,B 0,C 180,E1 -9818.327,E2 -9818.327} C_VEL
LIN {X 0,Y 424.965,Z 761.859,A -85,B 0,C 180,E1 -9819.759,E2 -9819.759} C_VEL
LIN {X 0,Y 425.488,Z 753.43,A -85,B 0,C 180,E1 -9821.191,E2 -9821.191} C_VEL
LIN {X 0,Y 426.133,Z 744.741,A -85,B 0,C 180,E1 -9822.38,E2 -9822.38} C_VEL
LIN {X 0,Y 426.829,Z 734.169,A -85,B 0,C 180,E1 -9823.556,E2 -9823.556} C_VEL
LIN {X 0,Y 427.466,Z 723.388,A -85,B 0,C 180,E1 -9824.52,E2 -9824.52} C_VEL
LIN {X 0,Y 428.139,Z 711.503,A -85,B 0,C 180,E1 -9825.348,E2 -9825.348} C_VEL
LIN {X 0,Y 428.707,Z 699.125,A -85,B 0,C 180,E1 -9825.998,E2 -9825.998} C_VEL
LIN {X 0,Y 429.254,Z 686.427,A -85,B 0,C 180,E1 -9826.466,E2 -9826.466} C_VEL
LIN {X 0,Y 429.564,Z 673.133,A -85,B 0,C 180,E1 -9826.759,E2 -9826.759} C_VEL
LIN {X 0,Y 430.197,Z 596.388,A -85,B 0,C 180,E1 -9828.042,E2 -9828.042} C_VEL
LIN {X 0,Y 426.587,Z 572.681,A -85,B 0,C 180,E1 -9828.613,E2 -9828.613} C_VEL
LIN {X 0,Y 427.622,Z 554.345,A -85,B 0,C 180,E1 -9832.21,E2 -9832.21} C_VEL
LIN {X 0,Y 428.101,Z 546.734,A -85,B 0,C 180,E1 -9833.716,E2 -9833.716} C_VEL
LIN {X 0,Y 426.353,Z 536.458,A -85,B 0,C 180,E1 -9835.901,E2 -9835.901} C_VEL
LIN {X 0,Y 425.376,Z 531.499,A -85,B 0,C 180,E1 -9837,E2 -9837} C_VEL
LIN {X 0,Y 425.29,Z 531.511,A -85,B 0,C 180,E1 -9839.719,E2 -9839.719} C_VEL
LIN {X 0,Y 425.281,Z 531.508,A -85,B 0,C 180,E1 -9843.047,E2 -9843.047} C_VEL
LIN {X 0,Y 425.281,Z 531.508,A -85,B 0,C 180,E1 -9845.928,E2 -9845.928} C_VEL
LIN {X 0,Y 425.3,Z 531.506,A -85,B 0,C 180,E1 -9849.044,E2 -9849.044} C_VEL
LIN {X 0,Y 425.274,Z 531.507,A -85,B 0,C 180,E1 -9852.652,E2 -9852.652} C_VEL
LIN {X 0,Y 425.257,Z 531.51,A -85,B 0,C 180,E1 -9856.043,E2 -9856.043} C_VEL
LIN {X 0,Y 425.299,Z 531.504,A -85,B 0,C 180,E1 -9858.624,E2 -9858.624} C_VEL
LIN {X 0,Y 425.318,Z 531.504,A -85,B 0,C 180,E1 -9861.103,E2 -9861.103} C_VEL
LIN {X 0,Y 425.294,Z 531.504,A -85,B 0,C 180,E1 -9864.664,E2 -9864.664} C_VEL
LIN {X 0,Y 425.259,Z 531.51,A -85,B 0,C 180,E1 -9868.073,E2 -9868.073} C_VEL
LIN {X 0,Y 425.331,Z 531.506,A -85,B 0,C 180,E1 -9871.368,E2 -9871.368} C_VEL
LIN {X 0,Y 425.287,Z 531.505,A -85,B 0,C 180,E1 -9874.554,E2 -9874.554} C_VEL
LIN {X 0,Y 425.28,Z 531.511,A -85,B 0,C 180,E1 -9877.661,E2 -9877.661} C_VEL
LIN {X 0,Y 425.353,Z 531.497,A -85,B 0,C 180,E1 -9880.704,E2 -9880.704} C_VEL
LIN {X 0,Y 425.379,Z 531.498,A -85,B 0,C 180,E1 -9883.688,E2 -9883.688} C_VEL
LIN {X 0,Y 425.403,Z 531.496,A -85,B 0,C 180,E1 -9887.598,E2 -9887.598} C_VEL
LIN {X 0,Y 425.433,Z 531.495,A -85,B 0,C 180,E1 -9891.45,E2 -9891.45} C_VEL
LIN {X 0,Y 425.545,Z 531.473,A -85,B 0,C 180,E1 -9894.313,E2 -9894.313} C_VEL
LIN {X 0,Y 425.566,Z 531.471,A -85,B 0,C 180,E1 -9898.107,E2 -9898.107} C_VEL
LIN {X 0,Y 425.693,Z 531.456,A -85,B 0,C 180,E1 -9900,E2 -9900} C_VEL
LIN {X 0,Y 425.55,Z 531.474,A -85,B 0,C 180,E1 -9902.84,E2 -9902.84} C_VEL
LIN {X 0,Y 425.523,Z 531.476,A -85,B 0,C 180,E1 -9906.641,E2 -9906.641} C_VEL
LIN {X 0,Y 425.393,Z 531.499,A -85,B 0,C 180,E1 -9909.51,E2 -9909.51} C_VEL
LIN {X 0,Y 425.385,Z 531.495,A -85,B 0,C 180,E1 -9912.904,E2 -9912.904} C_VEL
LIN {X 0,Y 425.353,Z 531.497,A -85,B 0,C 180,E1 -9916.605,E2 -9916.605} C_VEL
LIN {X 0,Y 425.321,Z 531.506,A -85,B 0,C 180,E1 -9919.636,E2 -9919.636} C_VEL
LIN {X 0,Y 425.3,Z 531.511,A -85,B 0,C 180,E1 -9923.366,E2 -9923.366} C_VEL
LIN {X 0,Y 425.342,Z 531.5,A -85,B 0,C 180,E1 -9926.845,E2 -9926.845} C_VEL
LIN {X 0,Y 425.312,Z 531.506,A -85,B 0,C 180,E1 -9929.718,E2 -9929.718} C_VEL
LIN {X 0,Y 425.277,Z 531.509,A -85,B 0,C 180,E1 -9933.049,E2 -9933.049} C_VEL
LIN {X 0,Y 425.279,Z 531.508,A -85,B 0,C 180,E1 -9935.93,E2 -9935.93} C_VEL
LIN {X 0,Y 425.299,Z 531.507,A -85,B 0,C 180,E1 -9939.045,E2 -9939.045} C_VEL
LIN {X 0,Y 425.275,Z 531.507,A -85,B 0,C 180,E1 -9942.654,E2 -9942.654} C_VEL
LIN {X 0,Y 425.316,Z 531.502,A -85,B 0,C 180,E1 -9946.053,E2 -9946.053} C_VEL
LIN {X 0,Y 425.308,Z 531.503,A -85,B 0,C 180,E1 -9948.627,E2 -9948.627} C_VEL
LIN {X 0,Y 425.322,Z 531.505,A -85,B 0,C 180,E1 -9951.105,E2 -9951.105} C_VEL
LIN {X 0,Y 425.3,Z 531.504,A -85,B 0,C 180,E1 -9954.665,E2 -9954.665} C_VEL
LIN {X 0,Y 425.265,Z 531.509,A -85,B 0,C 180,E1 -9958.074,E2 -9958.074} C_VEL
LIN {X 0,Y 425.332,Z 531.507,A -85,B 0,C 180,E1 -9961.369,E2 -9961.369} C_VEL
LIN {X 0,Y 425.296,Z 531.504,A -85,B 0,C 180,E1 -9964.555,E2 -9964.555} C_VEL
LIN {X 0,Y 425.29,Z 531.513,A -85,B 0,C 180,E1 -9967.662,E2 -9967.662} C_VEL
LIN {X 0,Y 425.422,Z 531.693,A -85,B 0,C 180,E1 -9971.02,E2 -9971.02} C_VEL
LIN {X 0,Y 427.045,Z 540.779,A -85,B 0,C 180,E1 -9973.272,E2 -9973.272} C_VEL
LIN {X 0,Y 426.929,Z 547.027,A -85,B 0,C 180,E1 -9974.729,E2 -9974.729} C_VEL
LIN {X 0,Y 426.783,Z 550.556,A -85,B 0,C 180,E1 -9975.487,E2 -9975.487} C_VEL
LIN {X 0,Y 430.478,Z 569.639,A -85,B 0,C 180,E1 -9975.968,E2 -9975.968} C_VEL
LIN {X 0,Y 429.545,Z 657.255,A -85,B 0,C 180,E1 -9977.45,E2 -9977.45} C_VEL
LIN {X 0,Y 429.168,Z 670.38,A -85,B 0,C 180,E1 -9977.859,E2 -9977.859} C_VEL
LIN {X 0,Y 428.648,Z 683.551,A -85,B 0,C 180,E1 -9978.474,E2 -9978.474} C_VEL
LIN {X 0,Y 428.071,Z 695.406,A -85,B 0,C 180,E1 -9979.237,E2 -9979.237} C_VEL
LIN {X 0,Y 427.441,Z 706.758,A -85,B 0,C 180,E1 -9980.178,E2 -9980.178} C_VEL
LIN {X 0,Y 427.016,Z 711.941,A -85,B 0,C 180,E1 -9980.684,E2 -9980.684} C_VEL
LIN {X 0,Y 426.021,Z 716.568,A -85,B 0,C 180,E1 -9981.159,E2 -9981.159} C_VEL
LIN {X 0,Y 422.768,Z 723.755,A -85,B 0,C 180,E1 -9981.969,E2 -9981.969} C_VEL
LIN {X 0,Y 419.561,Z 730.397,A -85,B 0,C 180,E1 -9982.868,E2 -9982.868} C_VEL
LIN {X 0,Y 418.647,Z 734.156,A -85,B 0,C 180,E1 -9983.477,E2 -9983.477} C_VEL
LIN {X 0,Y 418.1,Z 741.642,A -85,B 0,C 180,E1 -9984.937,E2 -9984.937} C_VEL
LIN {X 0,Y 417.632,Z 748.467,A -85,B 0,C 180,E1 -9986.623,E2 -9986.623} C_VEL
LIN {X 0,Y 417.225,Z 752.98,A -85,B 0,C 180,E1 -9988.069,E2 -9988.069} C_VEL
LIN {X 0,Y 417.112,Z 755.358,A -85,B 0,C 180,E1 -9989.035,E2 -9989.035} C_VEL
LIN {X 0,Y 417.044,Z 757.307,A -85,B 0,C 180,E1 -9990,E2 -9990} C_VEL
LIN {X 0,Y 417.035,Z 758.847,A -85,B 0,C 180,E1 -9990.966,E2 -9990.966} C_VEL
LIN {X 0,Y 417.076,Z 759.956,A -85,B 0,C 180,E1 -9991.931,E2 -9991.931} C_VEL
LIN {X 0,Y 417.059,Z 760.655,A -85,B 0,C 180,E1 -9992.898,E2 -9992.898} C_VEL
LIN {X 0,Y 417.055,Z 760.914,A -85,B 0,C 180,E1 -9994.833,E2 -9994.833} C_VEL
LIN {X 0,Y 417.085,Z 760.13,A -85,B 0,C 180,E1 -9996.187,E2 -9996.187} C_VEL
LIN {X 0,Y 417.117,Z 758.279,A -85,B 0,C 180,E1 -9997.746,E2 -9997.746} C_VEL
LIN {X 0,Y 417.25,Z 755.561,A -85,B 0,C 180,E1 -9999.207,E2 -9999.207} C_VEL
LIN {X 0,Y 417.462,Z 751.819,A -85,B 0,C 180,E1 -10000.672,E2 -10000.672} C_VEL
LIN {X 0,Y 417.788,Z 746.941,A -85,B 0,C 180,E1 -10002.138,E2 -10002.138} C_VEL
LIN {X 0,Y 418.211,Z 740.779,A -85,B 0,C 180,E1 -10003.607,E2 -10003.607} C_VEL
LIN {X 0,Y 418.863,Z 733.081,A -85,B 0,C 180,E1 -10005.074,E2 -10005.074} C_VEL
LIN {X 0,Y 419.521,Z 725.171,A -85,B 0,C 180,E1 -10006.296,E2 -10006.296} C_VEL
LIN {X 0,Y 420.27,Z 714.792,A -85,B 0,C 180,E1 -10007.599,E2 -10007.599} C_VEL
LIN {X 0,Y 421.011,Z 704.713,A -85,B 0,C 180,E1 -10008.617,E2 -10008.617} C_VEL
LIN {X 0,Y 421.741,Z 694.224,A -85,B 0,C 180,E1 -10009.468,E2 -10009.468} C_VEL
LIN {X 0,Y 422.427,Z 682.697,A -85,B 0,C 180,E1 -10010.195,E2 -10010.195} C_VEL
LIN {X 0,Y 422.952,Z 669.629,A -85,B 0,C 180,E1 -10010.804,E2 -10010.804} C_VEL
LIN {X 0,Y 423.358,Z 656.846,A -85,B 0,C 180,E1 -10011.197,E2 -10011.197} C_VEL
LIN {X 0,Y 424.384,Z 570.636,A -85,B 0,C 180,E1 -10012.685,E2 -10012.685} C_VEL
LIN {X 0,Y 420.167,Z 550.582,A -85,B 0,C 180,E1 -10013.262,E2 -10013.262} C_VEL
LIN {X 0,Y 420.48,Z 544.538,A -85,B 0,C 180,E1 -10014.699,E2 -10014.699} C_VEL
LIN {X 0,Y 419.046,Z 535.843,A -85,B 0,C 180,E1 -10016.925,E2 -10016.925} C_VEL
LIN {X 0,Y 418.326,Z 532.373,A -85,B 0,C 180,E1 -10017.878,E2 -10017.878} C_VEL
LIN {X 0,Y 418.212,Z 532.389,A -85,B 0,C 180,E1 -10021.395,E2 -10021.395} C_VEL
LIN {X 0,Y 418.265,Z 532.387,A -85,B 0,C 180,E1 -10024.579,E2 -10024.579} C_VEL
LIN {X 0,Y 418.237,Z 532.384,A -85,B 0,C 180,E1 -10027.834,E2 -10027.834} C_VEL
LIN {X 0,Y 418.265,Z 532.385,A -85,B 0,C 180,E1 -10030.942,E2 -10030.942} C_VEL
LIN {X 0,Y 418.266,Z 532.381,A -85,B 0,C 180,E1 -10033.737,E2 -10033.737} C_VEL
LIN {X 0,Y 418.213,Z 532.391,A -85,B 0,C 180,E1 -10036.449,E2 -10036.449} C_VEL
LIN {X 0,Y 418.261,Z 532.377,A -85,B 0,C 180,E1 -10039.123,E2 -10039.123} C_VEL
LIN {X 0,Y 418.231,Z 532.387,A -85,B 0,C 180,E1 -10042.164,E2 -10042.164} C_VEL
LIN {X 0,Y 418.261,Z 532.38,A -85,B 0,C 180,E1 -10045.419,E2 -10045.419} C_VEL
LIN {X 0,Y 418.213,Z 532.392,A -85,B 0,C 180,E1 -10048.604,E2 -10048.604} C_VEL
LIN {X 0,Y 418.289,Z 532.379,A -85,B 0,C 180,E1 -10051.936,E2 -10051.936} C_VEL
LIN {X 0,Y 418.283,Z 532.38,A -85,B 0,C 180,E1 -10055.162,E2 -10055.162} C_VEL
LIN {X 0,Y 418.226,Z 532.384,A -85,B 0,C 180,E1 -10058.303,E2 -10058.303} C_VEL
LIN {X 0,Y 418.275,Z 532.377,A -85,B 0,C 180,E1 -10061.383,E2 -10061.383} C_VEL
LIN {X 0,Y 418.294,Z 532.381,A -85,B 0,C 180,E1 -10064.405,E2 -10064.405} C_VEL
LIN {X 0,Y 418.347,Z 532.366,A -85,B 0,C 180,E1 -10067.385,E2 -10067.385} C_VEL
LIN {X 0,Y 418.333,Z 532.376,A -85,B 0,C 180,E1 -10070.328,E2 -10070.328} C_VEL
LIN {X 0,Y 418.485,Z 532.352,A -85,B 0,C 180,E1 -10073.249,E2 -10073.249} C_VEL
LIN {X 0,Y 418.334,Z 532.373,A -85,B 0,C 180,E1 -10075.181,E2 -10075.181} C_VEL
LIN {X 0,Y 418.536,Z 532.342,A -85,B 0,C 180,E1 -10078.075,E2 -10078.075} C_VEL
LIN {X 0,Y 418.665,Z 532.331,A -85,B 0,C 180,E1 -10080,E2 -10080} C_VEL
LIN {X 0,Y 418.503,Z 532.349,A -85,B 0,C 180,E1 -10082.888,E2 -10082.888} C_VEL
LIN {X 0,Y 418.484,Z 532.356,A -85,B 0,C 180,E1 -10086.751,E2 -10086.751} C_VEL
LIN {X 0,Y 418.333,Z 532.37,A -85,B 0,C 180,E1 -10089.671,E2 -10089.671} C_VEL
LIN {X 0,Y 418.337,Z 532.368,A -85,B 0,C 180,E1 -10093.001,E2 -10093.001} C_VEL
LIN {X 0,Y 418.304,Z 532.379,A -85,B 0,C 180,E1 -10096.736,E2 -10096.736} C_VEL
LIN {X 0,Y 418.262,Z 532.38,A -85,B 0,C 180,E1 -10099.791,E2 -10099.791} C_VEL
LIN {X 0,Y 418.224,Z 532.386,A -85,B 0,C 180,E1 -10102.737,E2 -10102.737} C_VEL
LIN {X 0,Y 418.263,Z 532.381,A -85,B 0,C 180,E1 -10105.905,E2 -10105.905} C_VEL
LIN {X 0,Y 418.267,Z 532.381,A -85,B 0,C 180,E1 -10109.162,E2 -10109.162} C_VEL
LIN {X 0,Y 418.251,Z 532.387,A -85,B 0,C 180,E1 -10112.845,E2 -10112.845} C_VEL
LIN {X 0,Y 418.243,Z 532.387,A -85,B 0,C 180,E1 -10116.239,E2 -10116.239} C_VEL
LIN {X 0,Y 418.26,Z 532.382,A -85,B 0,C 180,E1 -10119.681,E2 -10119.681} C_VEL
LIN {X 0,Y 418.24,Z 532.39,A -85,B 0,C 180,E1 -10122.324,E2 -10122.324} C_VEL
LIN {X 0,Y 418.235,Z 532.387,A -85,B 0,C 180,E1 -10125.11,E2 -10125.11} C_VEL
LIN {X 0,Y 418.239,Z 532.386,A -85,B 0,C 180,E1 -10127.768,E2 -10127.768} C_VEL
LIN {X 0,Y 418.257,Z 532.388,A -85,B 0,C 180,E1 -10130.619,E2 -10130.619} C_VEL
LIN {X 0,Y 418.243,Z 532.386,A -85,B 0,C 180,E1 -10133.977,E2 -10133.977} C_VEL
LIN {X 0,Y 418.256,Z 532.386,A -85,B 0,C 180,E1 -10137.157,E2 -10137.157} C_VEL
LIN {X 0,Y 418.268,Z 532.385,A -85,B 0,C 180,E1 -10140.896,E2 -10140.896} C_VEL
LIN {X 0,Y 418.361,Z 532.465,A -85,B 0,C 180,E1 -10142.247,E2 -10142.247} C_VEL
LIN {X 0,Y 421.138,Z 546.028,A -85,B 0,C 180,E1 -10145.343,E2 -10145.343} C_VEL
LIN {X 0,Y 421.531,Z 549.768,A -85,B 0,C 180,E1 -10146.153,E2 -10146.153} C_VEL
LIN {X 0,Y 420.394,Z 564.691,A -85,B 0,C 180,E1 -10149.192,E2 -10149.192} C_VEL
LIN {X 0,Y 419.935,Z 572.454,A -85,B 0,C 180,E1 -10150.761,E2 -10150.761} C_VEL
LIN {X 0,Y 424.045,Z 596.957,A -85,B 0,C 180,E1 -10151.407,E2 -10151.407} C_VEL
LIN {X 0,Y 423.234,Z 680.445,A -85,B 0,C 180,E1 -10152.858,E2 -10152.858} C_VEL
LIN {X 0,Y 422.648,Z 693.748,A -85,B 0,C 180,E1 -10153.269,E2 -10153.269} C_VEL
LIN {X 0,Y 422.064,Z 706.476,A -85,B 0,C 180,E1 -10153.867,E2 -10153.867} C_VEL
